LIN {X 0,Y 255.736,Z 943.824,A -85,B 0,C 180,E1 11654.094,E2 11654.094} C_VEL
LIN {X 0,Y 247.335,Z 955.504,A -85,B 0,C 180,E1 11649.69,E2 11649.69} C_VEL
LIN {X 0,Y 239.94,Z 965.687,A -85,B 0,C 180,E1 11644.807,E2 11644.807} C_VEL
LIN {X 0,Y 233.834,Z 974.598,A -85,B 0,C 180,E1 11639.45,E2 11639.45} C_VEL
LIN {X 0,Y 229.531,Z 981.362,A -85,B 0,C 180,E1 11634.168,E2 11634.168} C_VEL
LIN {X 0,Y 226.431,Z 987.137,A -85,B 0,C 180,E1 11628.268,E2 11628.268} C_VEL
LIN {X 0,Y 224.909,Z 990.729,A -85,B 0,C 180,E1 11623.102,E2 11623.102} C_VEL
LIN {X 0,Y 224.206,Z 993.296,A -85,B 0,C 180,E1 11617.687,E2 11617.687} C_VEL
LIN {X 0,Y 224.031,Z 994.4,A -85,B 0,C 180,E1 11612.557,E2 11612.557} C_VEL
LIN {X 0,Y 224.032,Z 994.473,A -85,B 0,C 180,E1 11608.209,E2 11608.209} C_VEL
LIN {X 0,Y 224.138,Z 993.662,A -85,B 0,C 180,E1 11603.597,E2 11603.597} C_VEL
LIN {X 0,Y 224.657,Z 991.562,A -85,B 0,C 180,E1 11598.187,E2 11598.187} C_VEL
LIN {X 0,Y 226.005,Z 988.015,A -85,B 0,C 180,E1 11592.759,E2 11592.759} C_VEL
LIN {X 0,Y 228.675,Z 982.95,A -85,B 0,C 180,E1 11587.101,E2 11587.101} C_VEL
LIN {X 0,Y 232.823,Z 976.112,A -85,B 0,C 180,E1 11581.533,E2 11581.533} C_VEL
LIN {X 0,Y 238.787,Z 967.412,A -85,B 0,C 180,E1 11576.004,E2 11576.004} C_VEL
LIN {X 0,Y 245.71,Z 957.743,A -85,B 0,C 180,E1 11571.2,E2 11571.2} C_VEL
LIN {X 0,Y 254.271,Z 945.935,A -85,B 0,C 180,E1 11566.522,E2 11566.522} C_VEL
LIN {X 0,Y 263.274,Z 933.388,A -85,B 0,C 180,E1 11562.533,E2 11562.533} C_VEL
LIN {X 0,Y 272.73,Z 919.575,A -85,B 0,C 180,E1 11559.001,E2 11559.001} C_VEL
LIN {X 0,Y 282.527,Z 904.622,A -85,B 0,C 180,E1 11555.871,E2 11555.871} C_VEL
LIN {X 0,Y 292.626,Z 887.873,A -85,B 0,C 180,E1 11553.047,E2 11553.047} C_VEL
LIN {X 0,Y 302.589,Z 870.047,A -85,B 0,C 180,E1 11550.589,E2 11550.589} C_VEL
LIN {X 0,Y 311.686,Z 851.804,A -85,B 0,C 180,E1 11548.554,E2 11548.554} C_VEL
LIN {X 0,Y 320.677,Z 831.7,A -85,B 0,C 180,E1 11546.722,E2 11546.722} C_VEL
LIN {X 0,Y 327.973,Z 812.96,A -85,B 0,C 180,E1 11545.336,E2 11545.336} C_VEL
LIN {X 0,Y 335.436,Z 790.655,A -85,B 0,C 180,E1 11544.005,E2 11544.005} C_VEL
LIN {X 0,Y 338.946,Z 778.487,A -85,B 0,C 180,E1 11543.397,E2 11543.397} C_VEL
LIN {X 0,Y 340.411,Z 771.364,A -85,B 0,C 180,E1 11542.929,E2 11542.929} C_VEL
LIN {X 0,Y 342.304,Z 753.795,A -85,B 0,C 180,E1 11541.314,E2 11541.314} C_VEL
LIN {X 0,Y 343.393,Z 746.488,A -85,B 0,C 180,E1 11540.937,E2 11540.937} C_VEL
LIN {X 0,Y 347.214,Z 723.354,A -85,B 0,C 180,E1 11540.335,E2 11540.335} C_VEL
LIN {X 0,Y 352.658,Z 665.576,A -85,B 0,C 180,E1 11539.208,E2 11539.208} C_VEL
LIN {X 0,Y 362.376,Z 558.402,A -85,B 0,C 180,E1 11537.172,E2 11537.172} C_VEL
LIN {X 0,Y 358.498,Z 551.455,A -85,B 0,C 180,E1 11534.455,E2 11534.455} C_VEL
LIN {X 0,Y 356.299,Z 547.697,A -85,B 0,C 180,E1 11532.644,E2 11532.644} C_VEL
LIN {X 0,Y 354.33,Z 544.268,A -85,B 0,C 180,E1 11530.734,E2 11530.734} C_VEL
LIN {X 0,Y 352.104,Z 540.388,A -85,B 0,C 180,E1 11527.999,E2 11527.999} C_VEL
LIN {X 0,Y 349.943,Z 536.182,A -85,B 0,C 180,E1 11523.44,E2 11523.44} C_VEL
LIN {X 0,Y 349.775,Z 535.565,A -85,B 0,C 180,E1 11522.622,E2 11522.622} C_VEL
LIN {X 0,Y 349.881,Z 535.803,A -85,B 0,C 180,E1 11517.38,E2 11517.38} C_VEL
LIN {X 0,Y 351.533,Z 539.751,A -85,B 0,C 180,E1 11513.304,E2 11513.304} C_VEL
LIN {X 0,Y 352.499,Z 541.08,A -85,B 0,C 180,E1 11511.929,E2 11511.929} C_VEL
LIN {X 0,Y 355.346,Z 546.022,A -85,B 0,C 180,E1 11508.723,E2 11508.723} C_VEL
LIN {X 0,Y 358.175,Z 550.942,A -85,B 0,C 180,E1 11506.274,E2 11506.274} C_VEL
LIN {X 0,Y 361.653,Z 557.016,A -85,B 0,C 180,E1 11503.786,E2 11503.786} C_VEL
LIN {X 0,Y 362.516,Z 559.023,A -85,B 0,C 180,E1 11503.197,E2 11503.197} C_VEL
LIN {X 0,Y 346.966,Z 729.479,A -85,B 0,C 180,E1 11499.934,E2 11499.934} C_VEL
LIN {X 0,Y 343.166,Z 753.522,A -85,B 0,C 180,E1 11499.355,E2 11499.355} C_VEL
LIN {X 0,Y 338.384,Z 775.393,A -85,B 0,C 180,E1 11498.689,E2 11498.689} C_VEL
LIN {X 0,Y 332.181,Z 797.399,A -85,B 0,C 180,E1 11497.784,E2 11497.784} C_VEL
LIN {X 0,Y 325.416,Z 817.772,A -85,B 0,C 180,E1 11496.722,E2 11496.722} C_VEL
LIN {X 0,Y 317.319,Z 838.274,A -85,B 0,C 180,E1 11495.361,E2 11495.361} C_VEL
LIN {X 0,Y 308.383,Z 858.36,A -85,B 0,C 180,E1 11493.712,E2 11493.712} C_VEL
LIN {X 0,Y 298.925,Z 877.022,A -85,B 0,C 180,E1 11491.796,E2 11491.796} C_VEL
LIN {X 0,Y 288.539,Z 895.73,A -85,B 0,C 180,E1 11489.432,E2 11489.432} C_VEL
LIN {X 0,Y 278.676,Z 911.928,A -85,B 0,C 180,E1 11486.896,E2 11486.896} C_VEL
LIN {X 0,Y 267.229,Z 929.456,A -85,B 0,C 180,E1 11483.494,E2 11483.494} C_VEL
LIN {X 0,Y 257.227,Z 944.006,A -85,B 0,C 180,E1 11479.967,E2 11479.967} C_VEL
LIN {X 0,Y 247.666,Z 957.322,A -85,B 0,C 180,E1 11475.934,E2 11475.934} C_VEL
LIN {X 0,Y 238.916,Z 969.495,A -85,B 0,C 180,E1 11471.388,E2 11471.388} C_VEL
LIN {X 0,Y 231.282,Z 980.172,A -85,B 0,C 180,E1 11466.314,E2 11466.314} C_VEL
LIN {X 0,Y 225.037,Z 989.575,A -85,B 0,C 180,E1 11460.724,E2 11460.724} C_VEL
LIN {X 0,Y 220.731,Z 996.778,A -85,B 0,C 180,E1 11455.199,E2 11455.199} C_VEL
LIN {X 0,Y 217.753,Z 1003.039,A -85,B 0,C 180,E1 11448.937,E2 11448.937} C_VEL
LIN {X 0,Y 216.47,Z 1006.872,A -85,B 0,C 180,E1 11443.624,E2 11443.624} C_VEL
LIN {X 0,Y 216.012,Z 1009.708,A -85,B 0,C 180,E1 11437.89,E2 11437.89} C_VEL
LIN {X 0,Y 216.005,Z 1010.89,A -85,B 0,C 180,E1 11432.654,E2 11432.654} C_VEL
LIN {X 0,Y 216.025,Z 1010.985,A -85,B 0,C 180,E1 11428.41,E2 11428.41} C_VEL
LIN {X 0,Y 216,Z 1010.188,A -85,B 0,C 180,E1 11423.89,E2 11423.89} C_VEL
LIN {X 0,Y 216.179,Z 1008.237,A -85,B 0,C 180,E1 11418.801,E2 11418.801} C_VEL
LIN {X 0,Y 217.196,Z 1004.462,A -85,B 0,C 180,E1 11412.868,E2 11412.868} C_VEL
LIN {X 0,Y 219.243,Z 999.668,A -85,B 0,C 180,E1 11407.479,E2 11407.479} C_VEL
LIN {X 0,Y 223.42,Z 992.094,A -85,B 0,C 180,E1 11401.102,E2 11401.102} C_VEL
LIN {X 0,Y 228.818,Z 983.779,A -85,B 0,C 180,E1 11395.675,E2 11395.675} C_VEL
LIN {X 0,Y 235.817,Z 973.673,A -85,B 0,C 180,E1 11390.504,E2 11390.504} C_VEL
LIN {X 0,Y 244.436,Z 961.795,A -85,B 0,C 180,E1 11385.623,E2 11385.623} C_VEL
LIN {X 0,Y 253.552,Z 949.029,A -85,B 0,C 180,E1 11381.483,E2 11381.483} C_VEL
LIN {X 0,Y 264.051,Z 934.069,A -85,B 0,C 180,E1 11377.563,E2 11377.563} C_VEL
LIN {X 0,Y 274.249,Z 918.722,A -85,B 0,C 180,E1 11374.344,E2 11374.344} C_VEL
LIN {X 0,Y 285.492,Z 900.645,A -85,B 0,C 180,E1 11371.303,E2 11371.303} C_VEL
LIN {X 0,Y 295.736,Z 882.842,A -85,B 0,C 180,E1 11368.89,E2 11368.89} C_VEL
LIN {X 0,Y 305.363,Z 864.194,A -85,B 0,C 180,E1 11366.862,E2 11366.862} C_VEL
LIN {X 0,Y 314.652,Z 844.373,A -85,B 0,C 180,E1 11365.106,E2 11365.106} C_VEL
LIN {X 0,Y 322.658,Z 824.612,A -85,B 0,C 180,E1 11363.711,E2 11363.711} C_VEL
LIN {X 0,Y 330.096,Z 803.74,A -85,B 0,C 180,E1 11362.523,E2 11362.523} C_VEL
LIN {X 0,Y 336.468,Z 781.982,A -85,B 0,C 180,E1 11361.564,E2 11361.564} C_VEL
LIN {X 0,Y 342.107,Z 758.231,A -85,B 0,C 180,E1 11360.78,E2 11360.78} C_VEL
LIN {X 0,Y 345.954,Z 736.026,A -85,B 0,C 180,E1 11360.221,E2 11360.221} C_VEL
LIN {X 0,Y 349.308,Z 704.022,A -85,B 0,C 180,E1 11359.57,E2 11359.57} C_VEL
LIN {X 0,Y 362.363,Z 558.559,A -85,B 0,C 180,E1 11356.783,E2 11356.783} C_VEL
LIN {X 0,Y 358.527,Z 551.667,A -85,B 0,C 180,E1 11354.123,E2 11354.123} C_VEL
LIN {X 0,Y 356.027,Z 547.407,A -85,B 0,C 180,E1 11352.076,E2 11352.076} C_VEL
LIN {X 0,Y 354.212,Z 544.29,A -85,B 0,C 180,E1 11350.325,E2 11350.325} C_VEL
LIN {X 0,Y 351.903,Z 540.251,A -85,B 0,C 180,E1 11347.51,E2 11347.51} C_VEL
LIN {X 0,Y 349.816,Z 536.268,A -85,B 0,C 180,E1 11343.277,E2 11343.277} C_VEL
LIN {X 0,Y 349.633,Z 535.518,A -85,B 0,C 180,E1 11342.458,E2 11342.458} C_VEL
LIN {X 0,Y 349.699,Z 535.594,A -85,B 0,C 180,E1 11336.721,E2 11336.721} C_VEL
LIN {X 0,Y 351.727,Z 540.075,A -85,B 0,C 180,E1 11332.157,E2 11332.157} C_VEL
LIN {X 0,Y 352.494,Z 541.282,A -85,B 0,C 180,E1 11331.107,E2 11331.107} C_VEL
LIN {X 0,Y 355.101,Z 545.709,A -85,B 0,C 180,E1 11328.221,E2 11328.221} C_VEL
LIN {X 0,Y 357.925,Z 550.622,A -85,B 0,C 180,E1 11325.769,E2 11325.769} C_VEL
LIN {X 0,Y 361.629,Z 557.156,A -85,B 0,C 180,E1 11323.123,E2 11323.123} C_VEL
LIN {X 0,Y 362.217,Z 558.605,A -85,B 0,C 180,E1 11322.717,E2 11322.717} C_VEL
LIN {X 0,Y 347.375,Z 720.612,A -85,B 0,C 180,E1 11319.623,E2 11319.623} C_VEL
LIN {X 0,Y 343.68,Z 744.239,A -85,B 0,C 180,E1 11319.029,E2 11319.029} C_VEL
LIN {X 0,Y 339.3,Z 764.96,A -85,B 0,C 180,E1 11318.331,E2 11318.331} C_VEL
LIN {X 0,Y 333.531,Z 786.231,A -85,B 0,C 180,E1 11317.399,E2 11317.399} C_VEL
LIN {X 0,Y 327.011,Z 806.35,A -85,B 0,C 180,E1 11316.295,E2 11316.295} C_VEL
LIN {X 0,Y 319.097,Z 826.901,A -85,B 0,C 180,E1 11314.883,E2 11314.883} C_VEL
LIN {X 0,Y 310.299,Z 846.954,A -85,B 0,C 180,E1 11313.183,E2 11313.183} C_VEL
LIN {X 0,Y 300.712,Z 865.928,A -85,B 0,C 180,E1 11311.176,E2 11311.176} C_VEL
LIN {X 0,Y 290.328,Z 884.559,A -85,B 0,C 180,E1 11308.752,E2 11308.752} C_VEL
LIN {X 0,Y 280.707,Z 900.187,A -85,B 0,C 180,E1 11306.243,E2 11306.243} C_VEL
LIN {X 0,Y 269.499,Z 917.069,A -85,B 0,C 180,E1 11302.898,E2 11302.898} C_VEL
LIN {X 0,Y 259.975,Z 930.527,A -85,B 0,C 180,E1 11299.588,E2 11299.588} C_VEL
LIN {X 0,Y 249.862,Z 944.136,A -85,B 0,C 180,E1 11295.414,E2 11295.414} C_VEL
LIN {X 0,Y 241.023,Z 955.816,A -85,B 0,C 180,E1 11290.947,E2 11290.947} C_VEL
LIN {X 0,Y 233.193,Z 965.999,A -85,B 0,C 180,E1 11285.968,E2 11285.968} C_VEL
LIN {X 0,Y 226.678,Z 974.909,A -85,B 0,C 180,E1 11280.476,E2 11280.476} C_VEL
LIN {X 0,Y 222.049,Z 981.671,A -85,B 0,C 180,E1 11275.037,E2 11275.037} C_VEL
LIN {X 0,Y 218.63,Z 987.551,A -85,B 0,C 180,E1 11268.795,E2 11268.795} C_VEL
LIN {X 0,Y 216.959,Z 991.187,A -85,B 0,C 180,E1 11263.32,E2 11263.32} C_VEL
LIN {X 0,Y 216.2,Z 993.743,A -85,B 0,C 180,E1 11257.439,E2 11257.439} C_VEL
LIN {X 0,Y 216.037,Z 994.721,A -85,B 0,C 180,E1 11252.386,E2 11252.386} C_VEL
LIN {X 0,Y 216.04,Z 994.751,A -85,B 0,C 180,E1 11247.878,E2 11247.878} C_VEL
LIN {X 0,Y 216.183,Z 993.835,A -85,B 0,C 180,E1 11242.826,E2 11242.826} C_VEL
LIN {X 0,Y 216.884,Z 991.406,A -85,B 0,C 180,E1 11236.945,E2 11236.945} C_VEL
LIN {X 0,Y 218.436,Z 987.924,A -85,B 0,C 180,E1 11231.59,E2 11231.59} C_VEL
LIN {X 0,Y 221.816,Z 982.087,A -85,B 0,C 180,E1 11225.218,E2 11225.218} C_VEL
LIN {X 0,Y 226.35,Z 975.393,A -85,B 0,C 180,E1 11219.766,E2 11219.766} C_VEL
LIN {X 0,Y 232.77,Z 966.624,A -85,B 0,C 180,E1 11214.258,E2 11214.258} C_VEL
LIN {X 0,Y 240.508,Z 956.545,A -85,B 0,C 180,E1 11209.26,E2 11209.26} C_VEL
LIN {X 0,Y 249.27,Z 944.999,A -85,B 0,C 180,E1 11204.773,E2 11204.773} C_VEL
LIN {X 0,Y 258.88,Z 932.201,A -85,B 0,C 180,E1 11200.748,E2 11200.748} C_VEL
LIN {X 0,Y 268.781,Z 918.217,A -85,B 0,C 180,E1 11197.251,E2 11197.251} C_VEL
LIN {X 0,Y 279.669,Z 902.002,A -85,B 0,C 180,E1 11193.968,E2 11193.968} C_VEL
LIN {X 0,Y 289.343,Z 886.364,A -85,B 0,C 180,E1 11191.411,E2 11191.411} C_VEL
LIN {X 0,Y 300.212,Z 867.107,A -85,B 0,C 180,E1 11188.856,E2 11188.856} C_VEL
LIN {X 0,Y 309.44,Z 848.964,A -85,B 0,C 180,E1 11186.911,E2 11186.911} C_VEL
LIN {X 0,Y 318.223,Z 829.319,A -85,B 0,C 180,E1 11185.203,E2 11185.203} C_VEL
LIN {X 0,Y 325.744,Z 810.262,A -85,B 0,C 180,E1 11183.851,E2 11183.851} C_VEL
LIN {X 0,Y 332.859,Z 788.912,A -85,B 0,C 180,E1 11182.635,E2 11182.635} C_VEL
LIN {X 0,Y 338.464,Z 768.92,A -85,B 0,C 180,E1 11181.725,E2 11181.725} C_VEL
LIN {X 0,Y 343.393,Z 746.488,A -85,B 0,C 180,E1 11180.937,E2 11180.937} C_VEL
LIN {X 0,Y 344.514,Z 739.093,A -85,B 0,C 180,E1 11180.585,E2 11180.585} C_VEL
LIN {X 0,Y 345.183,Z 720.8,A -85,B 0,C 180,E1 11179.191,E2 11179.191} C_VEL
LIN {X 0,Y 345.682,Z 713.298,A -85,B 0,C 180,E1 11178.876,E2 11178.876} C_VEL
LIN {X 0,Y 359.612,Z 563.719,A -85,B 0,C 180,E1 11176.046,E2 11176.046} C_VEL
LIN {X 0,Y 355.587,Z 556.366,A -85,B 0,C 180,E1 11172.918,E2 11172.918} C_VEL
LIN {X 0,Y 352.966,Z 551.864,A -85,B 0,C 180,E1 11170.363,E2 11170.363} C_VEL
LIN {X 0,Y 350.894,Z 548.153,A -85,B 0,C 180,E1 11167.697,E2 11167.697} C_VEL
LIN {X 0,Y 348.892,Z 543.886,A -85,B 0,C 180,E1 11163.122,E2 11163.122} C_VEL
LIN {X 0,Y 348.663,Z 543.461,A -85,B 0,C 180,E1 11161.972,E2 11161.972} C_VEL
LIN {X 0,Y 348.864,Z 543.694,A -85,B 0,C 180,E1 11157.536,E2 11157.536} C_VEL
LIN {X 0,Y 350.453,Z 547.629,A -85,B 0,C 180,E1 11153.447,E2 11153.447} C_VEL
LIN {X 0,Y 351.334,Z 548.905,A -85,B 0,C 180,E1 11152.149,E2 11152.149} C_VEL
LIN {X 0,Y 354.024,Z 553.722,A -85,B 0,C 180,E1 11149.01,E2 11149.01} C_VEL
LIN {X 0,Y 356.874,Z 558.835,A -85,B 0,C 180,E1 11146.471,E2 11146.471} C_VEL
LIN {X 0,Y 359.77,Z 564.022,A -85,B 0,C 180,E1 11144.326,E2 11144.326} C_VEL
LIN {X 0,Y 344.288,Z 729.198,A -85,B 0,C 180,E1 11141.191,E2 11141.191} C_VEL
LIN {X 0,Y 340.425,Z 753.168,A -85,B 0,C 180,E1 11140.625,E2 11140.625} C_VEL
LIN {X 0,Y 335.387,Z 775.727,A -85,B 0,C 180,E1 11139.951,E2 11139.951} C_VEL
LIN {X 0,Y 328.992,Z 797.784,A -85,B 0,C 180,E1 11139.057,E2 11139.057} C_VEL
LIN {X 0,Y 321.945,Z 818.389,A -85,B 0,C 180,E1 11137.995,E2 11137.995} C_VEL
LIN {X 0,Y 314.004,Z 837.972,A -85,B 0,C 180,E1 11136.715,E2 11136.715} C_VEL
LIN {X 0,Y 304.795,Z 858.143,A -85,B 0,C 180,E1 11135.086,E2 11135.086} C_VEL
LIN {X 0,Y 295.23,Z 876.513,A -85,B 0,C 180,E1 11133.229,E2 11133.229} C_VEL
LIN {X 0,Y 284.769,Z 894.861,A -85,B 0,C 180,E1 11130.948,E2 11130.948} C_VEL
LIN {X 0,Y 274.559,Z 911.107,A -85,B 0,C 180,E1 11128.437,E2 11128.437} C_VEL
LIN {X 0,Y 263.06,Z 928.159,A -85,B 0,C 180,E1 11125.175,E2 11125.175} C_VEL
LIN {X 0,Y 253.036,Z 942.127,A -85,B 0,C 180,E1 11121.837,E2 11121.837} C_VEL
LIN {X 0,Y 242.401,Z 956.361,A -85,B 0,C 180,E1 11117.584,E2 11117.584} C_VEL
LIN {X 0,Y 233.106,Z 968.597,A -85,B 0,C 180,E1 11112.995,E2 11112.995} C_VEL
LIN {X 0,Y 224.931,Z 979.388,A -85,B 0,C 180,E1 11107.834,E2 11107.834} C_VEL
LIN {X 0,Y 218.164,Z 988.898,A -85,B 0,C 180,E1 11102.113,E2 11102.113} C_VEL
LIN {X 0,Y 213.429,Z 996.154,A -85,B 0,C 180,E1 11096.424,E2 11096.424} C_VEL
LIN {X 0,Y 210.206,Z 1002.23,A -85,B 0,C 180,E1 11090.316,E2 11090.316} C_VEL
LIN {X 0,Y 208.596,Z 1006.399,A -85,B 0,C 180,E1 11084.432,E2 11084.432} C_VEL
LIN {X 0,Y 208.058,Z 1009.14,A -85,B 0,C 180,E1 11078.846,E2 11078.846} C_VEL
LIN {X 0,Y 208,Z 1010.54,A -85,B 0,C 180,E1 11073.307,E2 11073.307} C_VEL
LIN {X 0,Y 208.03,Z 1010.706,A -85,B 0,C 180,E1 11068.593,E2 11068.593} C_VEL
LIN {X 0,Y 208.003,Z 1009.958,A -85,B 0,C 180,E1 11063.931,E2 11063.931} C_VEL
LIN {X 0,Y 208.143,Z 1008.293,A -85,B 0,C 180,E1 11059.204,E2 11059.204} C_VEL
LIN {X 0,Y 209.127,Z 1004.799,A -85,B 0,C 180,E1 11053.046,E2 11053.046} C_VEL
LIN {X 0,Y 211.328,Z 999.885,A -85,B 0,C 180,E1 11047.175,E2 11047.175} C_VEL
LIN {X 0,Y 215.468,Z 992.874,A -85,B 0,C 180,E1 11040.845,E2 11040.845} C_VEL
LIN {X 0,Y 220.996,Z 984.741,A -85,B 0,C 180,E1 11035.251,E2 11035.251} C_VEL
LIN {X 0,Y 228.997,Z 973.899,A -85,B 0,C 180,E1 11029.422,E2 11029.422} C_VEL
LIN {X 0,Y 237.623,Z 962.61,A -85,B 0,C 180,E1 11024.643,E2 11024.643} C_VEL
LIN {X 0,Y 247.548,Z 949.427,A -85,B 0,C 180,E1 11020.246,E2 11020.246} C_VEL
LIN {X 0,Y 258.234,Z 934.926,A -85,B 0,C 180,E1 11016.365,E2 11016.365} C_VEL
LIN {X 0,Y 268.996,Z 919.346,A -85,B 0,C 180,E1 11013.063,E2 11013.063} C_VEL
LIN {X 0,Y 280.592,Z 901.455,A -85,B 0,C 180,E1 11010.027,E2 11010.027} C_VEL
LIN {X 0,Y 290.757,Z 884.374,A -85,B 0,C 180,E1 11007.701,E2 11007.701} C_VEL
LIN {X 0,Y 301.381,Z 864.601,A -85,B 0,C 180,E1 11005.542,E2 11005.542} C_VEL
LIN {X 0,Y 310.762,Z 845.178,A -85,B 0,C 180,E1 11003.832,E2 11003.832} C_VEL
LIN {X 0,Y 319.352,Z 824.613,A -85,B 0,C 180,E1 11002.395,E2 11002.395} C_VEL
LIN {X 0,Y 327.079,Z 803.428,A -85,B 0,C 180,E1 11001.212,E2 11001.212} C_VEL
LIN {X 0,Y 333.585,Z 781.67,A -85,B 0,C 180,E1 11000.275,E2 11000.275} C_VEL
LIN {X 0,Y 339.361,Z 757.786,A -85,B 0,C 180,E1 10999.506,E2 10999.506} C_VEL
LIN {X 0,Y 343.28,Z 735.546,A -85,B 0,C 180,E1 10998.956,E2 10998.956} C_VEL
LIN {X 0,Y 346.729,Z 703.302,A -85,B 0,C 180,E1 10998.308,E2 10998.308} C_VEL
LIN {X 0,Y 359.572,Z 563.811,A -85,B 0,C 180,E1 10995.648,E2 10995.648} C_VEL
LIN {X 0,Y 355.496,Z 556.371,A -85,B 0,C 180,E1 10992.507,E2 10992.507} C_VEL
LIN {X 0,Y 352.919,Z 551.985,A -85,B 0,C 180,E1 10990.034,E2 10990.034} C_VEL
LIN {X 0,Y 350.809,Z 548.129,A -85,B 0,C 180,E1 10987.368,E2 10987.368} C_VEL
LIN {X 0,Y 348.787,Z 544.163,A -85,B 0,C 180,E1 10983.122,E2 10983.122} C_VEL
LIN {X 0,Y 348.614,Z 543.445,A -85,B 0,C 180,E1 10982.301,E2 10982.301} C_VEL
LIN {X 0,Y 348.68,Z 543.493,A -85,B 0,C 180,E1 10976.876,E2 10976.876} C_VEL
LIN {X 0,Y 350.754,Z 548.075,A -85,B 0,C 180,E1 10972.135,E2 10972.135} C_VEL
LIN {X 0,Y 353.703,Z 553.253,A -85,B 0,C 180,E1 10968.587,E2 10968.587} C_VEL
LIN {X 0,Y 356.528,Z 558.35,A -85,B 0,C 180,E1 10966.043,E2 10966.043} C_VEL
LIN {X 0,Y 359.461,Z 563.796,A -85,B 0,C 180,E1 10963.843,E2 10963.843} C_VEL
LIN {X 0,Y 344.671,Z 720.935,A -85,B 0,C 180,E1 10960.869,E2 10960.869} C_VEL
LIN {X 0,Y 340.897,Z 744.553,A -85,B 0,C 180,E1 10960.285,E2 10960.285} C_VEL
LIN {X 0,Y 336.421,Z 765.272,A -85,B 0,C 180,E1 10959.601,E2 10959.601} C_VEL
LIN {X 0,Y 330.525,Z 786.54,A -85,B 0,C 180,E1 10958.686,E2 10958.686} C_VEL
LIN {X 0,Y 323.854,Z 806.66,A -85,B 0,C 180,E1 10957.601,E2 10957.601} C_VEL
LIN {X 0,Y 315.75,Z 827.211,A -85,B 0,C 180,E1 10956.211,E2 10956.211} C_VEL
LIN {X 0,Y 306.724,Z 847.263,A -85,B 0,C 180,E1 10954.535,E2 10954.535} C_VEL
LIN {X 0,Y 296.818,Z 866.336,A -85,B 0,C 180,E1 10952.541,E2 10952.541} C_VEL
LIN {X 0,Y 286.325,Z 884.625,A -85,B 0,C 180,E1 10950.188,E2 10950.188} C_VEL
LIN {X 0,Y 276.269,Z 900.441,A -85,B 0,C 180,E1 10947.668,E2 10947.668} C_VEL
LIN {X 0,Y 264.62,Z 917.38,A -85,B 0,C 180,E1 10944.318,E2 10944.318} C_VEL
LIN {X 0,Y 254.707,Z 930.839,A -85,B 0,C 180,E1 10941.001,E2 10941.001} C_VEL
LIN {X 0,Y 244.125,Z 944.448,A -85,B 0,C 180,E1 10936.797,E2 10936.797} C_VEL
LIN {X 0,Y 234.565,Z 956.47,A -85,B 0,C 180,E1 10932.124,E2 10932.124} C_VEL
LIN {X 0,Y 226.193,Z 966.758,A -85,B 0,C 180,E1 10926.948,E2 10926.948} C_VEL
LIN {X 0,Y 219.053,Z 975.904,A -85,B 0,C 180,E1 10921.045,E2 10921.045} C_VEL
LIN {X 0,Y 214.235,Z 982.567,A -85,B 0,C 180,E1 10915.424,E2 10915.424} C_VEL
LIN {X 0,Y 210.737,Z 988.147,A -85,B 0,C 180,E1 10909.107,E2 10909.107} C_VEL
LIN {X 0,Y 209.013,Z 991.644,A -85,B 0,C 180,E1 10903.554,E2 10903.554} C_VEL
LIN {X 0,Y 208.208,Z 994.109,A -85,B 0,C 180,E1 10897.448,E2 10897.448} C_VEL
LIN {X 0,Y 208.043,Z 995.021,A -85,B 0,C 180,E1 10892.478,E2 10892.478} C_VEL
LIN {X 0,Y 208.044,Z 995.051,A -85,B 0,C 180,E1 10887.796,E2 10887.796} C_VEL
LIN {X 0,Y 208.191,Z 994.2,A -85,B 0,C 180,E1 10882.827,E2 10882.827} C_VEL
LIN {X 0,Y 208.88,Z 992.015,A -85,B 0,C 180,E1 10876.999,E2 10876.999} C_VEL
LIN {X 0,Y 210.587,Z 988.428,A -85,B 0,C 180,E1 10871.165,E2 10871.165} C_VEL
LIN {X 0,Y 213.994,Z 982.98,A -85,B 0,C 180,E1 10864.84,E2 10864.84} C_VEL
LIN {X 0,Y 218.716,Z 976.386,A -85,B 0,C 180,E1 10859.205,E2 10859.205} C_VEL
LIN {X 0,Y 225.753,Z 967.38,A -85,B 0,C 180,E1 10853.283,E2 10853.283} C_VEL
LIN {X 0,Y 233.443,Z 957.859,A -85,B 0,C 180,E1 10848.409,E2 10848.409} C_VEL
LIN {X 0,Y 243.022,Z 945.929,A -85,B 0,C 180,E1 10843.611,E2 10843.611} C_VEL
LIN {X 0,Y 253.164,Z 933.047,A -85,B 0,C 180,E1 10839.484,E2 10839.484} C_VEL
LIN {X 0,Y 263.881,Z 918.523,A -85,B 0,C 180,E1 10835.829,E2 10835.829} C_VEL
LIN {X 0,Y 275.167,Z 902.307,A -85,B 0,C 180,E1 10832.551,E2 10832.551} C_VEL
LIN {X 0,Y 285.165,Z 886.667,A -85,B 0,C 180,E1 10830.009,E2 10830.009} C_VEL
LIN {X 0,Y 296.364,Z 867.408,A -85,B 0,C 180,E1 10827.476,E2 10827.476} C_VEL
LIN {X 0,Y 305.849,Z 849.264,A -85,B 0,C 180,E1 10825.554,E2 10825.554} C_VEL
LIN {X 0,Y 314.861,Z 829.617,A -85,B 0,C 180,E1 10823.87,E2 10823.87} C_VEL
LIN {X 0,Y 322.956,Z 809.561,A -85,B 0,C 180,E1 10822.475,E2 10822.475} C_VEL
LIN {X 0,Y 330.197,Z 788.07,A -85,B 0,C 180,E1 10821.289,E2 10821.289} C_VEL
LIN {X 0,Y 336.266,Z 766.6,A -85,B 0,C 180,E1 10820.349,E2 10820.349} C_VEL
LIN {X 0,Y 340.928,Z 745.163,A -85,B 0,C 180,E1 10819.633,E2 10819.633} C_VEL
LIN {X 0,Y 344.72,Z 721.844,A -85,B 0,C 180,E1 10819.05,E2 10819.05} C_VEL
LIN {X 0,Y 345.682,Z 713.298,A -85,B 0,C 180,E1 10818.876,E2 10818.876} C_VEL
LIN {X 0,Y 346.177,Z 705.769,A -85,B 0,C 180,E1 10818.575,E2 10818.575} C_VEL
LIN {X 0,Y 346.074,Z 686.167,A -85,B 0,C 180,E1 10817.216,E2 10817.216} C_VEL
LIN {X 0,Y 346.442,Z 679.68,A -85,B 0,C 180,E1 10816.971,E2 10816.971} C_VEL
LIN {X 0,Y 356.948,Z 569.278,A -85,B 0,C 180,E1 10814.897,E2 10814.897} C_VEL
LIN {X 0,Y 353.7,Z 563.225,A -85,B 0,C 180,E1 10812.158,E2 10812.158} C_VEL
LIN {X 0,Y 351.689,Z 559.561,A -85,B 0,C 180,E1 10810.07,E2 10810.07} C_VEL
LIN {X 0,Y 349.807,Z 556.031,A -85,B 0,C 180,E1 10807.556,E2 10807.556} C_VEL
LIN {X 0,Y 347.853,Z 551.589,A -85,B 0,C 180,E1 10802.801,E2 10802.801} C_VEL
LIN {X 0,Y 347.825,Z 551.442,A -85,B 0,C 180,E1 10797.859,E2 10797.859} C_VEL
LIN {X 0,Y 349.477,Z 555.634,A -85,B 0,C 180,E1 10793.429,E2 10793.429} C_VEL
LIN {X 0,Y 350.226,Z 556.864,A -85,B 0,C 180,E1 10792.289,E2 10792.289} C_VEL
LIN {X 0,Y 352.787,Z 561.578,A -85,B 0,C 180,E1 10789.219,E2 10789.219} C_VEL
LIN {X 0,Y 355.481,Z 566.551,A -85,B 0,C 180,E1 10786.748,E2 10786.748} C_VEL
LIN {X 0,Y 357.095,Z 569.815,A -85,B 0,C 180,E1 10785.455,E2 10785.455} C_VEL
LIN {X 0,Y 341.771,Z 728.983,A -85,B 0,C 180,E1 10782.467,E2 10782.467} C_VEL
LIN {X 0,Y 337.815,Z 753.006,A -85,B 0,C 180,E1 10781.909,E2 10781.909} C_VEL
LIN {X 0,Y 332.803,Z 775.066,A -85,B 0,C 180,E1 10781.266,E2 10781.266} C_VEL
LIN {X 0,Y 326.74,Z 795.771,A -85,B 0,C 180,E1 10780.461,E2 10780.461} C_VEL
LIN {X 0,Y 319.343,Z 817.176,A -85,B 0,C 180,E1 10779.401,E2 10779.401} C_VEL
LIN {X 0,Y 310.829,Z 837.76,A -85,B 0,C 180,E1 10778.091,E2 10778.091} C_VEL
LIN {X 0,Y 301.432,Z 857.84,A -85,B 0,C 180,E1 10776.5,E2 10776.5} C_VEL
LIN {X 0,Y 291.5,Z 876.412,A -85,B 0,C 180,E1 10774.652,E2 10774.652} C_VEL
LIN {X 0,Y 280.482,Z 895.116,A -85,B 0,C 180,E1 10772.345,E2 10772.345} C_VEL
LIN {X 0,Y 269.962,Z 911.312,A -85,B 0,C 180,E1 10769.851,E2 10769.851} C_VEL
LIN {X 0,Y 257.752,Z 928.707,A -85,B 0,C 180,E1 10766.505,E2 10766.505} C_VEL
LIN {X 0,Y 247.369,Z 942.599,A -85,B 0,C 180,E1 10763.152,E2 10763.152} C_VEL
LIN {X 0,Y 236.3,Z 956.696,A -85,B 0,C 180,E1 10758.859,E2 10758.859} C_VEL
LIN {X 0,Y 226.59,Z 968.869,A -85,B 0,C 180,E1 10754.197,E2 10754.197} C_VEL
LIN {X 0,Y 217.993,Z 979.546,A -85,B 0,C 180,E1 10748.926,E2 10748.926} C_VEL
LIN {X 0,Y 210.839,Z 988.95,A -85,B 0,C 180,E1 10743.046,E2 10743.046} C_VEL
LIN {X 0,Y 205.812,Z 996.157,A -85,B 0,C 180,E1 10737.169,E2 10737.169} C_VEL
LIN {X 0,Y 202.14,Z 1002.569,A -85,B 0,C 180,E1 10730.256,E2 10730.256} C_VEL
LIN {X 0,Y 200.587,Z 1006.428,A -85,B 0,C 180,E1 10724.431,E2 10724.431} C_VEL
LIN {X 0,Y 200.038,Z 1009.176,A -85,B 0,C 180,E1 10718.248,E2 10718.248} C_VEL
LIN {X 0,Y 200.01,Z 1010.289,A -85,B 0,C 180,E1 10712.866,E2 10712.866} C_VEL
LIN {X 0,Y 200.034,Z 1010.385,A -85,B 0,C 180,E1 10708.282,E2 10708.282} C_VEL
LIN {X 0,Y 200.009,Z 1009.656,A -85,B 0,C 180,E1 10703.687,E2 10703.687} C_VEL
LIN {X 0,Y 200.179,Z 1007.988,A -85,B 0,C 180,E1 10698.769,E2 10698.769} C_VEL
LIN {X 0,Y 201.292,Z 1004.491,A -85,B 0,C 180,E1 10692.365,E2 10692.365} C_VEL
LIN {X 0,Y 203.715,Z 999.573,A -85,B 0,C 180,E1 10686.271,E2 10686.271} C_VEL
LIN {X 0,Y 208.214,Z 992.56,A -85,B 0,C 180,E1 10679.725,E2 10679.725} C_VEL
LIN {X 0,Y 214.16,Z 984.425,A -85,B 0,C 180,E1 10673.972,E2 10673.972} C_VEL
LIN {X 0,Y 222.69,Z 973.583,A -85,B 0,C 180,E1 10668.017,E2 10668.017} C_VEL
LIN {X 0,Y 231.743,Z 962.362,A -85,B 0,C 180,E1 10663.193,E2 10663.193} C_VEL
LIN {X 0,Y 242.22,Z 949.111,A -85,B 0,C 180,E1 10658.733,E2 10658.733} C_VEL
LIN {X 0,Y 253.365,Z 934.609,A -85,B 0,C 180,E1 10654.842,E2 10654.842} C_VEL
LIN {X 0,Y 264.559,Z 919.013,A -85,B 0,C 180,E1 10651.548,E2 10651.548} C_VEL
LIN {X 0,Y 276.843,Z 900.663,A -85,B 0,C 180,E1 10648.472,E2 10648.472} C_VEL
LIN {X 0,Y 287.389,Z 883.446,A -85,B 0,C 180,E1 10646.169,E2 10646.169} C_VEL
LIN {X 0,Y 297.936,Z 864.289,A -85,B 0,C 180,E1 10644.118,E2 10644.118} C_VEL
LIN {X 0,Y 307.681,Z 844.605,A -85,B 0,C 180,E1 10642.42,E2 10642.42} C_VEL
LIN {X 0,Y 316.312,Z 824.382,A -85,B 0,C 180,E1 10641.038,E2 10641.038} C_VEL
LIN {X 0,Y 324.237,Z 803.117,A -85,B 0,C 180,E1 10639.878,E2 10639.878} C_VEL
LIN {X 0,Y 330.874,Z 781.358,A -85,B 0,C 180,E1 10638.963,E2 10638.963} C_VEL
LIN {X 0,Y 336.759,Z 757.472,A -85,B 0,C 180,E1 10638.215,E2 10638.215} C_VEL
LIN {X 0,Y 340.751,Z 735.228,A -85,B 0,C 180,E1 10637.676,E2 10637.676} C_VEL
LIN {X 0,Y 344.293,Z 702.888,A -85,B 0,C 180,E1 10637.034,E2 10637.034} C_VEL
LIN {X 0,Y 356.921,Z 569.404,A -85,B 0,C 180,E1 10634.52,E2 10634.52} C_VEL
LIN {X 0,Y 353.512,Z 563.08,A -85,B 0,C 180,E1 10631.667,E2 10631.667} C_VEL
LIN {X 0,Y 351.635,Z 559.68,A -85,B 0,C 180,E1 10629.74,E2 10629.74} C_VEL
LIN {X 0,Y 349.604,Z 555.883,A -85,B 0,C 180,E1 10627.064,E2 10627.064} C_VEL
LIN {X 0,Y 347.729,Z 551.865,A -85,B 0,C 180,E1 10622.801,E2 10622.801} C_VEL
LIN {X 0,Y 347.558,Z 551.359,A -85,B 0,C 180,E1 10621.978,E2 10621.978} C_VEL
LIN {X 0,Y 347.688,Z 551.588,A -85,B 0,C 180,E1 10616.867,E2 10616.867} C_VEL
LIN {X 0,Y 350.049,Z 556.661,A -85,B 0,C 180,E1 10611.706,E2 10611.706} C_VEL
LIN {X 0,Y 352.469,Z 561.116,A -85,B 0,C 180,E1 10608.795,E2 10608.795} C_VEL
LIN {X 0,Y 355.045,Z 565.897,A -85,B 0,C 180,E1 10606.399,E2 10606.399} C_VEL
LIN {X 0,Y 356.813,Z 569.323,A -85,B 0,C 180,E1 10604.98,E2 10604.98} C_VEL
LIN {X 0,Y 342.132,Z 721.258,A -85,B 0,C 180,E1 10602.135,E2 10602.135} C_VEL
LIN {X 0,Y 338.28,Z 744.866,A -85,B 0,C 180,E1 10601.562,E2 10601.562} C_VEL
LIN {X 0,Y 333.71,Z 765.584,A -85,B 0,C 180,E1 10600.892,E2 10600.892} C_VEL
LIN {X 0,Y 327.688,Z 786.85,A -85,B 0,C 180,E1 10599.996,E2 10599.996} C_VEL
LIN {X 0,Y 320.869,Z 806.969,A -85,B 0,C 180,E1 10598.932,E2 10598.932} C_VEL
LIN {X 0,Y 312.577,Z 827.52,A -85,B 0,C 180,E1 10597.567,E2 10597.567} C_VEL
LIN {X 0,Y 303.326,Z 847.572,A -85,B 0,C 180,E1 10595.918,E2 10595.918} C_VEL
LIN {X 0,Y 293.346,Z 866.299,A -85,B 0,C 180,E1 10593.993,E2 10593.993} C_VEL
LIN {X 0,Y 282.705,Z 884.387,A -85,B 0,C 180,E1 10591.708,E2 10591.708} C_VEL
LIN {X 0,Y 271.959,Z 900.769,A -85,B 0,C 180,E1 10589.125,E2 10589.125} C_VEL
LIN {X 0,Y 259.908,Z 917.692,A -85,B 0,C 180,E1 10585.791,E2 10585.791} C_VEL
LIN {X 0,Y 249.599,Z 931.15,A -85,B 0,C 180,E1 10582.472,E2 10582.472} C_VEL
LIN {X 0,Y 238.54,Z 944.761,A -85,B 0,C 180,E1 10578.245,E2 10578.245} C_VEL
LIN {X 0,Y 228.78,Z 956.441,A -85,B 0,C 180,E1 10573.664,E2 10573.664} C_VEL
LIN {X 0,Y 220.012,Z 966.623,A -85,B 0,C 180,E1 10568.5,E2 10568.5} C_VEL
LIN {X 0,Y 212.601,Z 975.531,A -85,B 0,C 180,E1 10562.736,E2 10562.736} C_VEL
LIN {X 0,Y 207.245,Z 982.291,A -85,B 0,C 180,E1 10556.965,E2 10556.965} C_VEL
LIN {X 0,Y 203.289,Z 988.059,A -85,B 0,C 180,E1 10550.436,E2 10550.436} C_VEL
LIN {X 0,Y 201.201,Z 991.796,A -85,B 0,C 180,E1 10544.385,E2 10544.385} C_VEL
LIN {X 0,Y 200.252,Z 994.347,A -85,B 0,C 180,E1 10538.035,E2 10538.035} C_VEL
LIN {X 0,Y 200.048,Z 995.321,A -85,B 0,C 180,E1 10532.577,E2 10532.577} C_VEL
LIN {X 0,Y 200.05,Z 995.372,A -85,B 0,C 180,E1 10527.994,E2 10527.994} C_VEL
LIN {X 0,Y 200.199,Z 994.565,A -85,B 0,C 180,E1 10522.827,E2 10522.827} C_VEL
LIN {X 0,Y 200.929,Z 992.472,A -85,B 0,C 180,E1 10516.768,E2 10516.768} C_VEL
LIN {X 0,Y 202.749,Z 988.931,A -85,B 0,C 180,E1 10510.708,E2 10510.708} C_VEL
LIN {X 0,Y 206.197,Z 983.851,A -85,B 0,C 180,E1 10504.413,E2 10504.413} C_VEL
LIN {X 0,Y 211.381,Z 977.037,A -85,B 0,C 180,E1 10498.332,E2 10498.332} C_VEL
LIN {X 0,Y 218.444,Z 968.583,A -85,B 0,C 180,E1 10492.504,E2 10492.504} C_VEL
LIN {X 0,Y 226.873,Z 958.67,A -85,B 0,C 180,E1 10487.263,E2 10487.263} C_VEL
LIN {X 0,Y 236.878,Z 946.859,A -85,B 0,C 180,E1 10482.388,E2 10482.388} C_VEL
LIN {X 0,Y 247.168,Z 934.346,A -85,B 0,C 180,E1 10478.307,E2 10478.307} C_VEL
LIN {X 0,Y 257.901,Z 920.493,A -85,B 0,C 180,E1 10474.732,E2 10474.732} C_VEL
LIN {X 0,Y 268.845,Z 905.535,A -85,B 0,C 180,E1 10471.616,E2 10471.616} C_VEL
LIN {X 0,Y 279.761,Z 889.163,A -85,B 0,C 180,E1 10468.892,E2 10468.892} C_VEL
LIN {X 0,Y 290.51,Z 871.669,A -85,B 0,C 180,E1 10466.523,E2 10466.523} C_VEL
LIN {X 0,Y 300.694,Z 852.906,A -85,B 0,C 180,E1 10464.493,E2 10464.493} C_VEL
LIN {X 0,Y 310.368,Z 832.936,A -85,B 0,C 180,E1 10462.742,E2 10462.742} C_VEL
LIN {X 0,Y 318.37,Z 813.847,A -85,B 0,C 180,E1 10461.397,E2 10461.397} C_VEL
LIN {X 0,Y 326.365,Z 791.535,A -85,B 0,C 180,E1 10460.132,E2 10460.132} C_VEL
LIN {X 0,Y 332.035,Z 772.449,A -85,B 0,C 180,E1 10459.275,E2 10459.275} C_VEL
LIN {X 0,Y 337.676,Z 748.701,A -85,B 0,C 180,E1 10458.447,E2 10458.447} C_VEL
LIN {X 0,Y 341.545,Z 726.722,A -85,B 0,C 180,E1 10457.883,E2 10457.883} C_VEL
LIN {X 0,Y 345.154,Z 693.391,A -85,B 0,C 180,E1 10457.228,E2 10457.228} C_VEL
LIN {X 0,Y 346.442,Z 679.68,A -85,B 0,C 180,E1 10456.971,E2 10456.971} C_VEL
LIN {X 0,Y 346.863,Z 672.143,A -85,B 0,C 180,E1 10456.668,E2 10456.668} C_VEL
LIN {X 0,Y 347.046,Z 652.551,A -85,B 0,C 180,E1 10455.312,E2 10455.312} C_VEL
LIN {X 0,Y 347.482,Z 646.068,A -85,B 0,C 180,E1 10455.072,E2 10455.072} C_VEL
LIN {X 0,Y 354.468,Z 574.884,A -85,B 0,C 180,E1 10453.76,E2 10453.76} C_VEL
LIN {X 0,Y 351.88,Z 570.048,A -85,B 0,C 180,E1 10451.39,E2 10451.39} C_VEL
LIN {X 0,Y 350.352,Z 567.151,A -85,B 0,C 180,E1 10449.694,E2 10449.694} C_VEL
LIN {X 0,Y 348.613,Z 563.792,A -85,B 0,C 180,E1 10447.25,E2 10447.25} C_VEL
LIN {X 0,Y 346.778,Z 559.365,A -85,B 0,C 180,E1 10442.314,E2 10442.314} C_VEL
LIN {X 0,Y 346.839,Z 559.477,A -85,B 0,C 180,E1 10437.853,E2 10437.853} C_VEL
LIN {X 0,Y 348.398,Z 563.511,A -85,B 0,C 180,E1 10433.574,E2 10433.574} C_VEL
LIN {X 0,Y 349.121,Z 564.816,A -85,B 0,C 180,E1 10432.43,E2 10432.43} C_VEL
LIN {X 0,Y 351.481,Z 569.275,A -85,B 0,C 180,E1 10429.511,E2 10429.511} C_VEL
LIN {X 0,Y 354.286,Z 574.603,A -85,B 0,C 180,E1 10426.869,E2 10426.869} C_VEL
LIN {X 0,Y 354.58,Z 575.378,A -85,B 0,C 180,E1 10426.605,E2 10426.605} C_VEL
LIN {X 0,Y 339.438,Z 728.661,A -85,B 0,C 180,E1 10423.763,E2 10423.763} C_VEL
LIN {X 0,Y 335.409,Z 752.687,A -85,B 0,C 180,E1 10423.217,E2 10423.217} C_VEL
LIN {X 0,Y 330.303,Z 774.774,A -85,B 0,C 180,E1 10422.59,E2 10422.59} C_VEL
LIN {X 0,Y 324.123,Z 795.475,A -85,B 0,C 180,E1 10421.809,E2 10421.809} C_VEL
LIN {X 0,Y 316.576,Z 816.878,A -85,B 0,C 180,E1 10420.777,E2 10420.777} C_VEL
LIN {X 0,Y 307.916,Z 837.372,A -85,B 0,C 180,E1 10419.506,E2 10419.506} C_VEL
LIN {X 0,Y 298.299,Z 857.462,A -85,B 0,C 180,E1 10417.951,E2 10417.951} C_VEL
LIN {X 0,Y 288.169,Z 875.934,A -85,B 0,C 180,E1 10416.151,E2 10416.151} C_VEL
LIN {X 0,Y 276.597,Z 895.024,A -85,B 0,C 180,E1 10413.832,E2 10413.832} C_VEL
LIN {X 0,Y 265.534,Z 911.517,A -85,B 0,C 180,E1 10411.314,E2 10411.314} C_VEL
LIN {X 0,Y 253.124,Z 928.559,A -85,B 0,C 180,E1 10408.042,E2 10408.042} C_VEL
LIN {X 0,Y 241.839,Z 943.072,A -85,B 0,C 180,E1 10404.527,E2 10404.527} C_VEL
LIN {X 0,Y 230.865,Z 956.383,A -85,B 0,C 180,E1 10400.428,E2 10400.428} C_VEL
LIN {X 0,Y 220.654,Z 968.556,A -85,B 0,C 180,E1 10395.715,E2 10395.715} C_VEL
LIN {X 0,Y 211.529,Z 979.232,A -85,B 0,C 180,E1 10390.354,E2 10390.354} C_VEL
LIN {X 0,Y 203.872,Z 988.637,A -85,B 0,C 180,E1 10384.329,E2 10384.329} C_VEL
LIN {X 0,Y 198.437,Z 995.845,A -85,B 0,C 180,E1 10378.268,E2 10378.268} C_VEL
LIN {X 0,Y 194.416,Z 1002.26,A -85,B 0,C 180,E1 10371.099,E2 10371.099} C_VEL
LIN {X 0,Y 192.711,Z 1006.033,A -85,B 0,C 180,E1 10365.199,E2 10365.199} C_VEL
LIN {X 0,Y 192.056,Z 1008.851,A -85,B 0,C 180,E1 10358.683,E2 10358.683} C_VEL
LIN {X 0,Y 192.013,Z 1009.989,A -85,B 0,C 180,E1 10352.985,E2 10352.985} C_VEL
LIN {X 0,Y 192.038,Z 1010.085,A -85,B 0,C 180,E1 10348.211,E2 10348.211} C_VEL
LIN {X 0,Y 192.009,Z 1009.354,A -85,B 0,C 180,E1 10343.423,E2 10343.423} C_VEL
LIN {X 0,Y 192.219,Z 1007.683,A -85,B 0,C 180,E1 10338.298,E2 10338.298} C_VEL
LIN {X 0,Y 193.481,Z 1004.182,A -85,B 0,C 180,E1 10331.628,E2 10331.628} C_VEL
LIN {X 0,Y 196.147,Z 999.262,A -85,B 0,C 180,E1 10325.296,E2 10325.296} C_VEL
LIN {X 0,Y 200.785,Z 992.61,A -85,B 0,C 180,E1 10318.814,E2 10318.814} C_VEL
LIN {X 0,Y 207.267,Z 984.315,A -85,B 0,C 180,E1 10312.745,E2 10312.745} C_VEL
LIN {X 0,Y 216.084,Z 973.794,A -85,B 0,C 180,E1 10306.786,E2 10306.786} C_VEL
LIN {X 0,Y 225.567,Z 962.632,A -85,B 0,C 180,E1 10301.876,E2 10301.876} C_VEL
LIN {X 0,Y 236.488,Z 949.508,A -85,B 0,C 180,E1 10297.368,E2 10297.368} C_VEL
LIN {X 0,Y 248.049,Z 935.132,A -85,B 0,C 180,E1 10293.458,E2 10293.458} C_VEL
LIN {X 0,Y 259.946,Z 919.186,A -85,B 0,C 180,E1 10290.08,E2 10290.08} C_VEL
LIN {X 0,Y 271.958,Z 901.951,A -85,B 0,C 180,E1 10287.176,E2 10287.176} C_VEL
LIN {X 0,Y 282.329,Z 885.593,A -85,B 0,C 180,E1 10284.974,E2 10284.974} C_VEL
LIN {X 0,Y 293.893,Z 865.46,A -85,B 0,C 180,E1 10282.801,E2 10282.801} C_VEL
LIN {X 0,Y 303.036,Z 847.564,A -85,B 0,C 180,E1 10281.254,E2 10281.254} C_VEL
LIN {X 0,Y 312.819,Z 825.701,A -85,B 0,C 180,E1 10279.748,E2 10279.748} C_VEL
LIN {X 0,Y 320.728,Z 805.157,A -85,B 0,C 180,E1 10278.632,E2 10278.632} C_VEL
LIN {X 0,Y 327.794,Z 782.944,A -85,B 0,C 180,E1 10277.699,E2 10277.699} C_VEL
LIN {X 0,Y 333.714,Z 760.164,A -85,B 0,C 180,E1 10276.981,E2 10276.981} C_VEL
LIN {X 0,Y 338.052,Z 737.028,A -85,B 0,C 180,E1 10276.424,E2 10276.424} C_VEL
LIN {X 0,Y 341.67,Z 706.223,A -85,B 0,C 180,E1 10275.813,E2 10275.813} C_VEL
LIN {X 0,Y 354.415,Z 574.964,A -85,B 0,C 180,E1 10273.375,E2 10273.375} C_VEL
LIN {X 0,Y 351.534,Z 569.588,A -85,B 0,C 180,E1 10270.737,E2 10270.737} C_VEL
LIN {X 0,Y 350.149,Z 567.05,A -85,B 0,C 180,E1 10269.201,E2 10269.201} C_VEL
LIN {X 0,Y 348.409,Z 563.632,A -85,B 0,C 180,E1 10266.757,E2 10266.757} C_VEL
LIN {X 0,Y 346.683,Z 559.566,A -85,B 0,C 180,E1 10262.479,E2 10262.479} C_VEL
LIN {X 0,Y 346.469,Z 559.255,A -85,B 0,C 180,E1 10258.015,E2 10258.015} C_VEL
LIN {X 0,Y 346.696,Z 559.676,A -85,B 0,C 180,E1 10256.859,E2 10256.859} C_VEL
LIN {X 0,Y 348.892,Z 564.484,A -85,B 0,C 180,E1 10251.927,E2 10251.927} C_VEL
LIN {X 0,Y 351.241,Z 568.975,A -85,B 0,C 180,E1 10249.005,E2 10249.005} C_VEL
LIN {X 0,Y 353.759,Z 573.797,A -85,B 0,C 180,E1 10246.599,E2 10246.599} C_VEL
LIN {X 0,Y 354.285,Z 575.067,A -85,B 0,C 180,E1 10246.13,E2 10246.13} C_VEL
LIN {X 0,Y 339.762,Z 721.588,A -85,B 0,C 180,E1 10243.419,E2 10243.419} C_VEL
LIN {X 0,Y 335.835,Z 745.18,A -85,B 0,C 180,E1 10242.857,E2 10242.857} C_VEL
LIN {X 0,Y 331.12,Z 766.11,A -85,B 0,C 180,E1 10242.195,E2 10242.195} C_VEL
LIN {X 0,Y 325.026,Z 787.16,A -85,B 0,C 180,E1 10241.327,E2 10241.327} C_VEL
LIN {X 0,Y 317.659,Z 808.401,A -85,B 0,C 180,E1 10240.222,E2 10240.222} C_VEL
LIN {X 0,Y 309.184,Z 828.721,A -85,B 0,C 180,E1 10238.884,E2 10238.884} C_VEL
LIN {X 0,Y 299.718,Z 848.635,A -85,B 0,C 180,E1 10237.263,E2 10237.263} C_VEL
LIN {X 0,Y 289.333,Z 867.55,A -85,B 0,C 180,E1 10235.333,E2 10235.333} C_VEL
LIN {X 0,Y 277.831,Z 886.342,A -85,B 0,C 180,E1 10232.947,E2 10232.947} C_VEL
LIN {X 0,Y 267.164,Z 902.063,A -85,B 0,C 180,E1 10230.461,E2 10230.461} C_VEL
LIN {X 0,Y 255.215,Z 918.205,A -85,B 0,C 180,E1 10227.272,E2 10227.272} C_VEL
LIN {X 0,Y 244.347,Z 931.86,A -85,B 0,C 180,E1 10223.896,E2 10223.896} C_VEL
LIN {X 0,Y 233.117,Z 945.073,A -85,B 0,C 180,E1 10219.761,E2 10219.761} C_VEL
LIN {X 0,Y 222.867,Z 956.753,A -85,B 0,C 180,E1 10215.133,E2 10215.133} C_VEL
LIN {X 0,Y 213.504,Z 967.039,A -85,B 0,C 180,E1 10209.822,E2 10209.822} C_VEL
LIN {X 0,Y 205.7,Z 975.842,A -85,B 0,C 180,E1 10203.98,E2 10203.98} C_VEL
LIN {X 0,Y 199.942,Z 982.6,A -85,B 0,C 180,E1 10198.034,E2 10198.034} C_VEL
LIN {X 0,Y 195.636,Z 988.366,A -85,B 0,C 180,E1 10191.273,E2 10191.273} C_VEL
LIN {X 0,Y 193.345,Z 992.101,A -85,B 0,C 180,E1 10184.983,E2 10184.983} C_VEL
LIN {X 0,Y 192.289,Z 994.649,A -85,B 0,C 180,E1 10178.37,E2 10178.37} C_VEL
LIN {X 0,Y 192.053,Z 995.621,A -85,B 0,C 180,E1 10172.684,E2 10172.684} C_VEL
LIN {X 0,Y 192.055,Z 995.672,A -85,B 0,C 180,E1 10167.911,E2 10167.911} C_VEL
LIN {X 0,Y 192.205,Z 994.931,A -85,B 0,C 180,E1 10162.828,E2 10162.828} C_VEL
LIN {X 0,Y 192.921,Z 993.041,A -85,B 0,C 180,E1 10156.819,E2 10156.819} C_VEL
LIN {X 0,Y 194.924,Z 989.435,A -85,B 0,C 180,E1 10150.213,E2 10150.213} C_VEL
LIN {X 0,Y 198.622,Z 984.39,A -85,B 0,C 180,E1 10143.644,E2 10143.644} C_VEL
LIN {X 0,Y 204.097,Z 977.688,A -85,B 0,C 180,E1 10137.396,E2 10137.396} C_VEL
LIN {X 0,Y 211.554,Z 969.339,A -85,B 0,C 180,E1 10131.405,E2 10131.405} C_VEL
LIN {X 0,Y 220.398,Z 959.482,A -85,B 0,C 180,E1 10126.05,E2 10126.05} C_VEL
LIN {X 0,Y 231.379,Z 947.168,A -85,B 0,C 180,E1 10120.874,E2 10120.874} C_VEL
LIN {X 0,Y 242.14,Z 934.653,A -85,B 0,C 180,E1 10116.775,E2 10116.775} C_VEL
LIN {X 0,Y 253.304,Z 920.798,A -85,B 0,C 180,E1 10113.203,E2 10113.203} C_VEL
LIN {X 0,Y 264.635,Z 905.84,A -85,B 0,C 180,E1 10110.102,E2 10110.102} C_VEL
LIN {X 0,Y 275.909,Z 889.454,A -85,B 0,C 180,E1 10107.402,E2 10107.402} C_VEL
LIN {X 0,Y 286.962,Z 871.97,A -85,B 0,C 180,E1 10105.066,E2 10105.066} C_VEL
LIN {X 0,Y 297.17,Z 853.675,A -85,B 0,C 180,E1 10103.115,E2 10103.115} C_VEL
LIN {X 0,Y 306.693,Z 834.677,A -85,B 0,C 180,E1 10101.461,E2 10101.461} C_VEL
LIN {X 0,Y 315.111,Z 815.141,A -85,B 0,C 180,E1 10100.096,E2 10100.096} C_VEL
LIN {X 0,Y 322.867,Z 794.382,A -85,B 0,C 180,E1 10098.919,E2 10098.919} C_VEL
LIN {X 0,Y 329.055,Z 774.213,A -85,B 0,C 180,E1 10098.015,E2 10098.015} C_VEL
LIN {X 0,Y 334.784,Z 751.19,A -85,B 0,C 180,E1 10097.209,E2 10097.209} C_VEL
LIN {X 0,Y 338.836,Z 729.079,A -85,B 0,C 180,E1 10096.642,E2 10096.642} C_VEL
LIN {X 0,Y 342.429,Z 698.232,A -85,B 0,C 180,E1 10096.035,E2 10096.035} C_VEL
LIN {X 0,Y 347.482,Z 646.068,A -85,B 0,C 180,E1 10095.072,E2 10095.072} C_VEL
LIN {X 0,Y 347.965,Z 638.531,A -85,B 0,C 180,E1 10094.774,E2 10094.774} C_VEL
LIN {X 0,Y 348.407,Z 618.954,A -85,B 0,C 180,E1 10093.418,E2 10093.418} C_VEL
LIN {X 0,Y 348.886,Z 612.473,A -85,B 0,C 180,E1 10093.178,E2 10093.178} C_VEL
LIN {X 0,Y 352.081,Z 580.67,A -85,B 0,C 180,E1 10092.59,E2 10092.59} C_VEL
LIN {X 0,Y 349.232,Z 575.06,A -85,B 0,C 180,E1 10089.559,E2 10089.559} C_VEL
LIN {X 0,Y 347.429,Z 571.55,A -85,B 0,C 180,E1 10086.943,E2 10086.943} C_VEL
LIN {X 0,Y 345.77,Z 567.295,A -85,B 0,C 180,E1 10082.155,E2 10082.155} C_VEL
LIN {X 0,Y 345.848,Z 567.553,A -85,B 0,C 180,E1 10077.847,E2 10077.847} C_VEL
LIN {X 0,Y 347.421,Z 571.518,A -85,B 0,C 180,E1 10073.556,E2 10073.556} C_VEL
LIN {X 0,Y 349.835,Z 576.189,A -85,B 0,C 180,E1 10070.209,E2 10070.209} C_VEL
LIN {X 0,Y 352.201,Z 580.97,A -85,B 0,C 180,E1 10067.777,E2 10067.777} C_VEL
LIN {X 0,Y 337.268,Z 728.456,A -85,B 0,C 180,E1 10065.074,E2 10065.074} C_VEL
LIN {X 0,Y 333.188,Z 752.335,A -85,B 0,C 180,E1 10064.543,E2 10064.543} C_VEL
LIN {X 0,Y 328.06,Z 774.169,A -85,B 0,C 180,E1 10063.944,E2 10063.944} C_VEL
LIN {X 0,Y 321.689,Z 795.18,A -85,B 0,C 180,E1 10063.178,E2 10063.178} C_VEL
LIN {X 0,Y 313.995,Z 816.58,A -85,B 0,C 180,E1 10062.177,E2 10062.177} C_VEL
LIN {X 0,Y 305.05,Z 837.3,A -85,B 0,C 180,E1 10060.926,E2 10060.926} C_VEL
LIN {X 0,Y 294.872,Z 857.976,A -85,B 0,C 180,E1 10059.353,E2 10059.353} C_VEL
LIN {X 0,Y 284.445,Z 876.477,A -85,B 0,C 180,E1 10057.575,E2 10057.575} C_VEL
LIN {X 0,Y 272.056,Z 896.186,A -85,B 0,C 180,E1 10055.186,E2 10055.186} C_VEL
LIN {X 0,Y 260.564,Z 912.748,A -85,B 0,C 180,E1 10052.653,E2 10052.653} C_VEL
LIN {X 0,Y 248.167,Z 929.062,A -85,B 0,C 180,E1 10049.493,E2 10049.493} C_VEL
LIN {X 0,Y 236.456,Z 943.544,A -85,B 0,C 180,E1 10045.966,E2 10045.966} C_VEL
LIN {X 0,Y 225.044,Z 956.719,A -85,B 0,C 180,E1 10041.843,E2 10041.843} C_VEL
LIN {X 0,Y 214.38,Z 968.789,A -85,B 0,C 180,E1 10037.069,E2 10037.069} C_VEL
LIN {X 0,Y 204.785,Z 979.39,A -85,B 0,C 180,E1 10031.602,E2 10031.602} C_VEL
LIN {X 0,Y 196.372,Z 989.054,A -85,B 0,C 180,E1 10025.121,E2 10025.121} C_VEL
LIN {X 0,Y 190.681,Z 996.162,A -85,B 0,C 180,E1 10018.84,E2 10018.84} C_VEL
LIN {X 0,Y 186.601,Z 1002.167,A -85,B 0,C 180,E1 10011.697,E2 10011.697} C_VEL
LIN {X 0,Y 184.732,Z 1005.984,A -85,B 0,C 180,E1 10005.379,E2 10005.379} C_VEL
LIN {X 0,Y 184.051,Z 1008.695,A -85,B 0,C 180,E1 9998.434,E2 9998.434} C_VEL
LIN {X 0,Y 184.016,Z 1009.689,A -85,B 0,C 180,E1 9993.115,E2 9993.115} C_VEL
LIN {X 0,Y 184.042,Z 1009.785,A -85,B 0,C 180,E1 9988.133,E2 9988.133} C_VEL
LIN {X 0,Y 184.007,Z 1009.052,A -85,B 0,C 180,E1 9983.136,E2 9983.136} C_VEL
LIN {X 0,Y 184.288,Z 1007.298,A -85,B 0,C 180,E1 9977.575,E2 9977.575} C_VEL
LIN {X 0,Y 185.797,Z 1003.658,A -85,B 0,C 180,E1 9970.513,E2 9970.513} C_VEL
LIN {X 0,Y 188.633,Z 998.949,A -85,B 0,C 180,E1 9964.241,E2 9964.241} C_VEL
LIN {X 0,Y 193.689,Z 992.296,A -85,B 0,C 180,E1 9957.535,E2 9957.535} C_VEL
LIN {X 0,Y 200.471,Z 984.211,A -85,B 0,C 180,E1 9951.438,E2 9951.438} C_VEL
LIN {X 0,Y 209.582,Z 974.005,A -85,B 0,C 180,E1 9945.476,E2 9945.476} C_VEL
LIN {X 0,Y 219.518,Z 962.902,A -85,B 0,C 180,E1 9940.487,E2 9940.487} C_VEL
LIN {X 0,Y 231.497,Z 949.192,A -85,B 0,C 180,E1 9935.72,E2 9935.72} C_VEL
LIN {X 0,Y 243.543,Z 934.817,A -85,B 0,C 180,E1 9931.818,E2 9931.818} C_VEL
LIN {X 0,Y 255.882,Z 918.871,A -85,B 0,C 180,E1 9928.469,E2 9928.469} C_VEL
LIN {X 0,Y 268.28,Z 901.637,A -85,B 0,C 180,E1 9925.604,E2 9925.604} C_VEL
LIN {X 0,Y 278.949,Z 885.28,A -85,B 0,C 180,E1 9923.439,E2 9923.439} C_VEL
LIN {X 0,Y 290.813,Z 865.148,A -85,B 0,C 180,E1 9921.311,E2 9921.311} C_VEL
LIN {X 0,Y 300.173,Z 847.252,A -85,B 0,C 180,E1 9919.801,E2 9919.801} C_VEL
LIN {X 0,Y 309.745,Z 826.401,A -85,B 0,C 180,E1 9918.393,E2 9918.393} C_VEL
LIN {X 0,Y 317.714,Z 806.216,A -85,B 0,C 180,E1 9917.315,E2 9917.315} C_VEL
LIN {X 0,Y 325.117,Z 783.705,A -85,B 0,C 180,E1 9916.383,E2 9916.383} C_VEL
LIN {X 0,Y 331.184,Z 761.034,A -85,B 0,C 180,E1 9915.68,E2 9915.68} C_VEL
LIN {X 0,Y 335.705,Z 737.687,A -85,B 0,C 180,E1 9915.128,E2 9915.128} C_VEL
LIN {X 0,Y 339.026,Z 711.385,A -85,B 0,C 180,E1 9914.606,E2 9914.606} C_VEL
LIN {X 0,Y 352.02,Z 580.793,A -85,B 0,C 180,E1 9912.216,E2 9912.216} C_VEL
LIN {X 0,Y 349.235,Z 575.28,A -85,B 0,C 180,E1 9909.309,E2 9909.309} C_VEL
LIN {X 0,Y 347.327,Z 571.51,A -85,B 0,C 180,E1 9906.612,E2 9906.612} C_VEL
LIN {X 0,Y 345.609,Z 567.241,A -85,B 0,C 180,E1 9901.989,E2 9901.989} C_VEL
LIN {X 0,Y 345.657,Z 567.381,A -85,B 0,C 180,E1 9897.181,E2 9897.181} C_VEL
LIN {X 0,Y 347.741,Z 572.306,A -85,B 0,C 180,E1 9892.15,E2 9892.15} C_VEL
LIN {X 0,Y 349.946,Z 576.676,A -85,B 0,C 180,E1 9889.297,E2 9889.297} C_VEL
LIN {X 0,Y 351.917,Z 580.67,A -85,B 0,C 180,E1 9887.298,E2 9887.298} C_VEL
LIN {X 0,Y 337.566,Z 721.919,A -85,B 0,C 180,E1 9884.72,E2 9884.72} C_VEL
LIN {X 0,Y 333.548,Z 745.564,A -85,B 0,C 180,E1 9884.17,E2 9884.17} C_VEL
LIN {X 0,Y 328.704,Z 766.638,A -85,B 0,C 180,E1 9883.518,E2 9883.518} C_VEL
LIN {X 0,Y 322.543,Z 787.47,A -85,B 0,C 180,E1 9882.68,E2 9882.68} C_VEL
LIN {X 0,Y 315.023,Z 808.711,A -85,B 0,C 180,E1 9881.601,E2 9881.601} C_VEL
LIN {X 0,Y 306.366,Z 829.03,A -85,B 0,C 180,E1 9880.294,E2 9880.294} C_VEL
LIN {X 0,Y 296.788,Z 848.744,A -85,B 0,C 180,E1 9878.725,E2 9878.725} C_VEL
LIN {X 0,Y 286.033,Z 867.859,A -85,B 0,C 180,E1 9876.813,E2 9876.813} C_VEL
LIN {X 0,Y 274.213,Z 886.652,A -85,B 0,C 180,E1 9874.467,E2 9874.467} C_VEL
LIN {X 0,Y 263.143,Z 902.478,A -85,B 0,C 180,E1 9871.996,E2 9871.996} C_VEL
LIN {X 0,Y 250.425,Z 919.057,A -85,B 0,C 180,E1 9868.731,E2 9868.731} C_VEL
LIN {X 0,Y 238.66,Z 933.288,A -85,B 0,C 180,E1 9865.188,E2 9865.188} C_VEL
LIN {X 0,Y 227.296,Z 946.007,A -85,B 0,C 180,E1 9861.124,E2 9861.124} C_VEL
LIN {X 0,Y 216.605,Z 957.598,A -85,B 0,C 180,E1 9856.438,E2 9856.438} C_VEL
LIN {X 0,Y 206.839,Z 967.748,A -85,B 0,C 180,E1 9851.052,E2 9851.052} C_VEL
LIN {X 0,Y 198.13,Z 976.941,A -85,B 0,C 180,E1 9844.656,E2 9844.656} C_VEL
LIN {X 0,Y 192.046,Z 983.706,A -85,B 0,C 180,E1 9838.372,E2 9838.372} C_VEL
LIN {X 0,Y 187.572,Z 989.267,A -85,B 0,C 180,E1 9831.249,E2 9831.249} C_VEL
LIN {X 0,Y 185.268,Z 992.864,A -85,B 0,C 180,E1 9824.691,E2 9824.691} C_VEL
LIN {X 0,Y 184.27,Z 995.078,A -85,B 0,C 180,E1 9818.108,E2 9818.108} C_VEL
LIN {X 0,Y 184.059,Z 995.922,A -85,B 0,C 180,E1 9812.801,E2 9812.801} C_VEL
LIN {X 0,Y 184.06,Z 995.972,A -85,B 0,C 180,E1 9807.82,E2 9807.82} C_VEL
LIN {X 0,Y 184.225,Z 995.232,A -85,B 0,C 180,E1 9802.516,E2 9802.516} C_VEL
LIN {X 0,Y 185.034,Z 993.344,A -85,B 0,C 180,E1 9796.246,E2 9796.246} C_VEL
LIN {X 0,Y 187.251,Z 989.741,A -85,B 0,C 180,E1 9789.366,E2 9789.366} C_VEL
LIN {X 0,Y 191.234,Z 984.746,A -85,B 0,C 180,E1 9782.609,E2 9782.609} C_VEL
LIN {X 0,Y 197.181,Z 977.997,A -85,B 0,C 180,E1 9776.101,E2 9776.101} C_VEL
LIN {X 0,Y 205.263,Z 969.521,A -85,B 0,C 180,E1 9769.887,E2 9769.887} C_VEL
LIN {X 0,Y 214.516,Z 959.79,A -85,B 0,C 180,E1 9764.515,E2 9764.515} C_VEL
LIN {X 0,Y 226.316,Z 947.183,A -85,B 0,C 180,E1 9759.181,E2 9759.181} C_VEL
LIN {X 0,Y 237.919,Z 934.272,A -85,B 0,C 180,E1 9754.974,E2 9754.974} C_VEL
LIN {X 0,Y 249.846,Z 919.919,A -85,B 0,C 180,E1 9751.349,E2 9751.349} C_VEL
LIN {X 0,Y 262.034,Z 904.219,A -85,B 0,C 180,E1 9748.195,E2 9748.195} C_VEL
LIN {X 0,Y 273.347,Z 888.125,A -85,B 0,C 180,E1 9745.636,E2 9745.636} C_VEL
LIN {X 0,Y 285.529,Z 868.971,A -85,B 0,C 180,E1 9743.203,E2 9743.203} C_VEL
LIN {X 0,Y 295.764,Z 850.891,A -85,B 0,C 180,E1 9741.368,E2 9741.368} C_VEL
LIN {X 0,Y 305.848,Z 830.509,A -85,B 0,C 180,E1 9739.71,E2 9739.71} C_VEL
LIN {X 0,Y 314.503,Z 810.448,A -85,B 0,C 180,E1 9738.399,E2 9738.399} C_VEL
LIN {X 0,Y 322.142,Z 789.195,A -85,B 0,C 180,E1 9737.299,E2 9737.299} C_VEL
LIN {X 0,Y 328.609,Z 767.72,A -85,B 0,C 180,E1 9736.42,E2 9736.42} C_VEL
LIN {X 0,Y 333.625,Z 746.024,A -85,B 0,C 180,E1 9735.744,E2 9735.744} C_VEL
LIN {X 0,Y 337.647,Z 722.678,A -85,B 0,C 180,E1 9735.196,E2 9735.196} C_VEL
LIN {X 0,Y 347.58,Z 625.438,A -85,B 0,C 180,E1 9733.411,E2 9733.411} C_VEL
LIN {X 0,Y 348.886,Z 612.473,A -85,B 0,C 180,E1 9733.178,E2 9733.178} C_VEL
LIN {X 0,Y 349.163,Z 607.477,A -85,B 0,C 180,E1 9732.923,E2 9732.923} C_VEL
LIN {X 0,Y 349.126,Z 595.074,A -85,B 0,C 180,E1 9731.7,E2 9731.7} C_VEL
LIN {X 0,Y 349.423,Z 590.761,A -85,B 0,C 180,E1 9731.502,E2 9731.502} C_VEL
LIN {X 0,Y 349.837,Z 586.486,A -85,B 0,C 180,E1 9731.401,E2 9731.401} C_VEL
LIN {X 0,Y 347.852,Z 582.541,A -85,B 0,C 180,E1 9729.096,E2 9729.096} C_VEL
LIN {X 0,Y 346.353,Z 579.429,A -85,B 0,C 180,E1 9726.798,E2 9726.798} C_VEL
LIN {X 0,Y 344.765,Z 575.224,A -85,B 0,C 180,E1 9721.995,E2 9721.995} C_VEL
LIN {X 0,Y 344.839,Z 575.444,A -85,B 0,C 180,E1 9718.006,E2 9718.006} C_VEL
LIN {X 0,Y 346.445,Z 579.521,A -85,B 0,C 180,E1 9713.538,E2 9713.538} C_VEL
LIN {X 0,Y 348.896,Z 584.668,A -85,B 0,C 180,E1 9710.099,E2 9710.099} C_VEL
LIN {X 0,Y 349.941,Z 586.956,A -85,B 0,C 180,E1 9708.947,E2 9708.947} C_VEL
LIN {X 0,Y 335.276,Z 728.251,A -85,B 0,C 180,E1 9706.402,E2 9706.402} C_VEL
LIN {X 0,Y 331.133,Z 752.052,A -85,B 0,C 180,E1 9705.885,E2 9705.885} C_VEL
LIN {X 0,Y 325.844,Z 774.187,A -85,B 0,C 180,E1 9705.296,E2 9705.296} C_VEL
LIN {X 0,Y 319.441,Z 794.884,A -85,B 0,C 180,E1 9704.568,E2 9704.568} C_VEL
LIN {X 0,Y 311.597,Z 816.302,A -85,B 0,C 180,E1 9703.598,E2 9703.598} C_VEL
LIN {X 0,Y 302.431,Z 837.11,A -85,B 0,C 180,E1 9702.379,E2 9702.379} C_VEL
LIN {X 0,Y 292.084,Z 857.673,A -85,B 0,C 180,E1 9700.856,E2 9700.856} C_VEL
LIN {X 0,Y 281.409,Z 876.172,A -85,B 0,C 180,E1 9699.124,E2 9699.124} C_VEL
LIN {X 0,Y 268.511,Z 896.137,A -85,B 0,C 180,E1 9696.753,E2 9696.753} C_VEL
LIN {X 0,Y 256.483,Z 912.953,A -85,B 0,C 180,E1 9694.214,E2 9694.214} C_VEL
LIN {X 0,Y 244.136,Z 928.636,A -85,B 0,C 180,E1 9691.205,E2 9691.205} C_VEL
LIN {X 0,Y 231.882,Z 943.233,A -85,B 0,C 180,E1 9687.678,E2 9687.678} C_VEL
LIN {X 0,Y 219.367,Z 957.054,A -85,B 0,C 180,E1 9683.333,E2 9683.333} C_VEL
LIN {X 0,Y 207.707,Z 969.53,A -85,B 0,C 180,E1 9678.251,E2 9678.251} C_VEL
LIN {X 0,Y 198.146,Z 979.548,A -85,B 0,C 180,E1 9672.934,E2 9672.934} C_VEL
LIN {X 0,Y 189.245,Z 989.106,A -85,B 0,C 180,E1 9666.277,E2 9666.277} C_VEL
LIN {X 0,Y 183.183,Z 996.164,A -85,B 0,C 180,E1 9659.779,E2 9659.779} C_VEL
LIN {X 0,Y 178.811,Z 1002.074,A -85,B 0,C 180,E1 9652.347,E2 9652.347} C_VEL
LIN {X 0,Y 176.788,Z 1005.845,A -85,B 0,C 180,E1 9645.751,E2 9645.751} C_VEL
LIN {X 0,Y 176.057,Z 1008.466,A -85,B 0,C 180,E1 9638.491,E2 9638.491} C_VEL
LIN {X 0,Y 176.024,Z 1009.413,A -85,B 0,C 180,E1 9632.931,E2 9632.931} C_VEL
LIN {X 0,Y 176.045,Z 1009.485,A -85,B 0,C 180,E1 9628.048,E2 9628.048} C_VEL
LIN {X 0,Y 176.009,Z 1008.75,A -85,B 0,C 180,E1 9622.822,E2 9622.822} C_VEL
LIN {X 0,Y 176.322,Z 1007.073,A -85,B 0,C 180,E1 9617.226,E2 9617.226} C_VEL
LIN {X 0,Y 177.937,Z 1003.564,A -85,B 0,C 180,E1 9609.958,E2 9609.958} C_VEL
LIN {X 0,Y 181.185,Z 998.637,A -85,B 0,C 180,E1 9603.099,E2 9603.099} C_VEL
LIN {X 0,Y 186.791,Z 991.87,A -85,B 0,C 180,E1 9596.065,E2 9596.065} C_VEL
LIN {X 0,Y 193.987,Z 983.895,A -85,B 0,C 180,E1 9589.895,E2 9589.895} C_VEL
LIN {X 0,Y 203.735,Z 973.622,A -85,B 0,C 180,E1 9583.786,E2 9583.786} C_VEL
LIN {X 0,Y 214.168,Z 962.585,A -85,B 0,C 180,E1 9578.781,E2 9578.781} C_VEL
LIN {X 0,Y 226.708,Z 948.875,A -85,B 0,C 180,E1 9574,E2 9574} C_VEL
LIN {X 0,Y 239.399,Z 934.323,A -85,B 0,C 180,E1 9570.078,E2 9570.078} C_VEL
LIN {X 0,Y 252.027,Z 918.557,A -85,B 0,C 180,E1 9566.808,E2 9566.808} C_VEL
LIN {X 0,Y 264.808,Z 901.323,A -85,B 0,C 180,E1 9563.989,E2 9563.989} C_VEL
LIN {X 0,Y 275.775,Z 884.967,A -85,B 0,C 180,E1 9561.868,E2 9561.868} C_VEL
LIN {X 0,Y 287.934,Z 864.836,A -85,B 0,C 180,E1 9559.791,E2 9559.791} C_VEL
LIN {X 0,Y 297.501,Z 846.952,A -85,B 0,C 180,E1 9558.323,E2 9558.323} C_VEL
LIN {X 0,Y 307.277,Z 826.09,A -85,B 0,C 180,E1 9556.955,E2 9556.955} C_VEL
LIN {X 0,Y 315.051,Z 806.808,A -85,B 0,C 180,E1 9555.952,E2 9555.952} C_VEL
LIN {X 0,Y 322.713,Z 784.136,A -85,B 0,C 180,E1 9555.034,E2 9555.034} C_VEL
LIN {X 0,Y 328.716,Z 762.212,A -85,B 0,C 180,E1 9554.371,E2 9554.371} C_VEL
LIN {X 0,Y 333.478,Z 738.668,A -85,B 0,C 180,E1 9553.822,E2 9553.822} C_VEL
LIN {X 0,Y 336.74,Z 714.504,A -85,B 0,C 180,E1 9553.345,E2 9553.345} C_VEL
LIN {X 0,Y 349.776,Z 586.573,A -85,B 0,C 180,E1 9551.041,E2 9551.041} C_VEL
LIN {X 0,Y 347.709,Z 582.543,A -85,B 0,C 180,E1 9548.683,E2 9548.683} C_VEL
LIN {X 0,Y 346.147,Z 579.257,A -85,B 0,C 180,E1 9546.301,E2 9546.301} C_VEL
LIN {X 0,Y 344.598,Z 575.169,A -85,B 0,C 180,E1 9541.829,E2 9541.829} C_VEL
LIN {X 0,Y 344.646,Z 575.276,A -85,B 0,C 180,E1 9537.339,E2 9537.339} C_VEL
LIN {X 0,Y 346.643,Z 580.256,A -85,B 0,C 180,E1 9532.292,E2 9532.292} C_VEL
LIN {X 0,Y 348.66,Z 584.376,A -85,B 0,C 180,E1 9529.591,E2 9529.591} C_VEL
LIN {X 0,Y 349.66,Z 586.632,A -85,B 0,C 180,E1 9528.476,E2 9528.476} C_VEL
LIN {X 0,Y 335.546,Z 722.245,A -85,B 0,C 180,E1 9526.038,E2 9526.038} C_VEL
LIN {X 0,Y 331.469,Z 745.807,A -85,B 0,C 180,E1 9525.503,E2 9525.503} C_VEL
LIN {X 0,Y 326.519,Z 766.95,A -85,B 0,C 180,E1 9524.868,E2 9524.868} C_VEL
LIN {X 0,Y 319.857,Z 788.929,A -85,B 0,C 180,E1 9524.001,E2 9524.001} C_VEL
LIN {X 0,Y 312.153,Z 810.109,A -85,B 0,C 180,E1 9522.942,E2 9522.942} C_VEL
LIN {X 0,Y 303.32,Z 830.231,A -85,B 0,C 180,E1 9521.666,E2 9521.666} C_VEL
LIN {X 0,Y 293.422,Z 849.979,A -85,B 0,C 180,E1 9520.114,E2 9520.114} C_VEL
LIN {X 0,Y 282.93,Z 868.168,A -85,B 0,C 180,E1 9518.327,E2 9518.327} C_VEL
LIN {X 0,Y 270.886,Z 886.831,A -85,B 0,C 180,E1 9516.045,E2 9516.045} C_VEL
LIN {X 0,Y 259.473,Z 902.684,A -85,B 0,C 180,E1 9513.612,E2 9513.612} C_VEL
LIN {X 0,Y 246.879,Z 918.626,A -85,B 0,C 180,E1 9510.533,E2 9510.533} C_VEL
LIN {X 0,Y 235.352,Z 932.086,A -85,B 0,C 180,E1 9507.253,E2 9507.253} C_VEL
LIN {X 0,Y 222.801,Z 945.696,A -85,B 0,C 180,E1 9503.006,E2 9503.006} C_VEL
LIN {X 0,Y 211.513,Z 957.378,A -85,B 0,C 180,E1 9498.314,E2 9498.314} C_VEL
LIN {X 0,Y 201.179,Z 967.559,A -85,B 0,C 180,E1 9492.906,E2 9492.906} C_VEL
LIN {X 0,Y 192.224,Z 976.464,A -85,B 0,C 180,E1 9486.733,E2 9486.733} C_VEL
LIN {X 0,Y 185.568,Z 983.22,A -85,B 0,C 180,E1 9480.425,E2 9480.425} C_VEL
LIN {X 0,Y 180.29,Z 989.18,A -85,B 0,C 180,E1 9472.839,E2 9472.839} C_VEL
LIN {X 0,Y 177.69,Z 992.712,A -85,B 0,C 180,E1 9466.338,E2 9466.338} C_VEL
LIN {X 0,Y 176.383,Z 995.253,A -85,B 0,C 180,E1 9459.131,E2 9459.131} C_VEL
LIN {X 0,Y 176.065,Z 996.222,A -85,B 0,C 180,E1 9452.928,E2 9452.928} C_VEL
LIN {X 0,Y 176.066,Z 996.272,A -85,B 0,C 180,E1 9447.721,E2 9447.721} C_VEL
LIN {X 0,Y 176.25,Z 995.534,A -85,B 0,C 180,E1 9442.175,E2 9442.175} C_VEL
LIN {X 0,Y 177.165,Z 993.648,A -85,B 0,C 180,E1 9435.623,E2 9435.623} C_VEL
LIN {X 0,Y 179.665,Z 989.982,A -85,B 0,C 180,E1 9428.339,E2 9428.339} C_VEL
LIN {X 0,Y 184.205,Z 984.795,A -85,B 0,C 180,E1 9421.115,E2 9421.115} C_VEL
LIN {X 0,Y 190.718,Z 977.964,A -85,B 0,C 180,E1 9414.417,E2 9414.417} C_VEL
LIN {X 0,Y 199.312,Z 969.51,A -85,B 0,C 180,E1 9408.153,E2 9408.153} C_VEL
LIN {X 0,Y 209.017,Z 959.883,A -85,B 0,C 180,E1 9402.788,E2 9402.788} C_VEL
LIN {X 0,Y 220.909,Z 947.784,A -85,B 0,C 180,E1 9397.628,E2 9397.628} C_VEL
LIN {X 0,Y 232.639,Z 935.267,A -85,B 0,C 180,E1 9393.518,E2 9393.518} C_VEL
LIN {X 0,Y 245.206,Z 920.775,A -85,B 0,C 180,E1 9389.833,E2 9389.833} C_VEL
LIN {X 0,Y 257.53,Z 905.52,A -85,B 0,C 180,E1 9386.762,E2 9386.762} C_VEL
LIN {X 0,Y 269.528,Z 888.976,A -85,B 0,C 180,E1 9384.15,E2 9384.15} C_VEL
LIN {X 0,Y 281.63,Z 870.594,A -85,B 0,C 180,E1 9381.829,E2 9381.829} C_VEL
LIN {X 0,Y 292.148,Z 852.54,A -85,B 0,C 180,E1 9380.014,E2 9380.014} C_VEL
LIN {X 0,Y 302.801,Z 831.7,A -85,B 0,C 180,E1 9378.335,E2 9378.335} C_VEL
LIN {X 0,Y 311.628,Z 811.742,A -85,B 0,C 180,E1 9377.053,E2 9377.053} C_VEL
LIN {X 0,Y 319.718,Z 789.862,A -85,B 0,C 180,E1 9375.941,E2 9375.941} C_VEL
LIN {X 0,Y 326.186,Z 768.904,A -85,B 0,C 180,E1 9375.102,E2 9375.102} C_VEL
LIN {X 0,Y 331.405,Z 746.96,A -85,B 0,C 180,E1 9374.429,E2 9374.429} C_VEL
LIN {X 0,Y 335.52,Z 723.917,A -85,B 0,C 180,E1 9373.896,E2 9373.896} C_VEL
LIN {X 0,Y 343.076,Z 652.384,A -85,B 0,C 180,E1 9372.596,E2 9372.596} C_VEL
LIN {X 0,Y 349.423,Z 590.761,A -85,B 0,C 180,E1 9371.502,E2 9371.502} C_VEL
LIN {X 0,Y 349.42,Z 588.796,A -85,B 0,C 180,E1 9371.294,E2 9371.294} C_VEL
LIN {X 0,Y 349.012,Z 587.534,A -85,B 0,C 180,E1 9370.809,E2 9370.809} C_VEL
LIN {X 0,Y 348.135,Z 587.41,A -85,B 0,C 180,E1 9369.99,E2 9369.99} C_VEL
LIN {X 0,Y 346.253,Z 588.966,A -85,B 0,C 180,E1 9368.202,E2 9368.202} C_VEL
LIN {X 0,Y 345.819,Z 588.568,A -85,B 0,C 180,E1 9367.607,E2 9367.607} C_VEL
LIN {X 0,Y 345.093,Z 587.051,A -85,B 0,C 180,E1 9366.321,E2 9366.321} C_VEL
LIN {X 0,Y 343.791,Z 583.165,A -85,B 0,C 180,E1 9362,E2 9362} C_VEL
LIN {X 0,Y 343.833,Z 583.335,A -85,B 0,C 180,E1 9358.167,E2 9358.167} C_VEL
LIN {X 0,Y 345.588,Z 588.009,A -85,B 0,C 180,E1 9353.271,E2 9353.271} C_VEL
LIN {X 0,Y 347.618,Z 592.363,A -85,B 0,C 180,E1 9350.397,E2 9350.397} C_VEL
LIN {X 0,Y 347.812,Z 593.038,A -85,B 0,C 180,E1 9350.137,E2 9350.137} C_VEL
LIN {X 0,Y 333.473,Z 727.996,A -85,B 0,C 180,E1 9347.745,E2 9347.745} C_VEL
LIN {X 0,Y 329.238,Z 751.879,A -85,B 0,C 180,E1 9347.241,E2 9347.241} C_VEL
LIN {X 0,Y 323.666,Z 774.707,A -85,B 0,C 180,E1 9346.651,E2 9346.651} C_VEL
LIN {X 0,Y 316.94,Z 795.878,A -85,B 0,C 180,E1 9345.924,E2 9345.924} C_VEL
LIN {X 0,Y 308.807,Z 817.406,A -85,B 0,C 180,E1 9344.968,E2 9344.968} C_VEL
LIN {X 0,Y 299.794,Z 837.378,A -85,B 0,C 180,E1 9343.827,E2 9343.827} C_VEL
LIN {X 0,Y 289.077,Z 858.111,A -85,B 0,C 180,E1 9342.326,E2 9342.326} C_VEL
LIN {X 0,Y 278.171,Z 876.542,A -85,B 0,C 180,E1 9340.636,E2 9340.636} C_VEL
LIN {X 0,Y 265.139,Z 896.135,A -85,B 0,C 180,E1 9338.352,E2 9338.352} C_VEL
LIN {X 0,Y 252.594,Z 913.165,A -85,B 0,C 180,E1 9335.823,E2 9335.823} C_VEL
LIN {X 0,Y 239.504,Z 929.184,A -85,B 0,C 180,E1 9332.763,E2 9332.763} C_VEL
LIN {X 0,Y 226.836,Z 943.673,A -85,B 0,C 180,E1 9329.25,E2 9329.25} C_VEL
LIN {X 0,Y 214.467,Z 956.742,A -85,B 0,C 180,E1 9325.129,E2 9325.129} C_VEL
LIN {X 0,Y 202.102,Z 969.324,A -85,B 0,C 180,E1 9319.974,E2 9319.974} C_VEL
LIN {X 0,Y 191.622,Z 979.706,A -85,B 0,C 180,E1 9314.357,E2 9314.357} C_VEL
LIN {X 0,Y 182.562,Z 988.793,A -85,B 0,C 180,E1 9307.832,E2 9307.832} C_VEL
LIN {X 0,Y 175.999,Z 995.853,A -85,B 0,C 180,E1 9301.127,E2 9301.127} C_VEL
LIN {X 0,Y 171.2,Z 1001.765,A -85,B 0,C 180,E1 9293.398,E2 9293.398} C_VEL
LIN {X 0,Y 168.915,Z 1005.55,A -85,B 0,C 180,E1 9286.482,E2 9286.482} C_VEL
LIN {X 0,Y 168.069,Z 1008.163,A -85,B 0,C 180,E1 9278.898,E2 9278.898} C_VEL
LIN {X 0,Y 168.027,Z 1009.113,A -85,B 0,C 180,E1 9273.071,E2 9273.071} C_VEL
LIN {X 0,Y 168.047,Z 1009.184,A -85,B 0,C 180,E1 9267.955,E2 9267.955} C_VEL
LIN {X 0,Y 168.017,Z 1008.447,A -85,B 0,C 180,E1 9262.479,E2 9262.479} C_VEL
LIN {X 0,Y 168.44,Z 1006.646,A -85,B 0,C 180,E1 9256.267,E2 9256.267} C_VEL
LIN {X 0,Y 170.465,Z 1002.822,A -85,B 0,C 180,E1 9248.317,E2 9248.317} C_VEL
LIN {X 0,Y 174.056,Z 998.046,A -85,B 0,C 180,E1 9241.509,E2 9241.509} C_VEL
LIN {X 0,Y 180.811,Z 990.573,A -85,B 0,C 180,E1 9233.729,E2 9233.729} C_VEL
LIN {X 0,Y 188.984,Z 982.287,A -85,B 0,C 180,E1 9227.341,E2 9227.341} C_VEL
LIN {X 0,Y 199.515,Z 971.789,A -85,B 0,C 180,E1 9221.269,E2 9221.269} C_VEL
LIN {X 0,Y 210.801,Z 960.51,A -85,B 0,C 180,E1 9216.271,E2 9216.271} C_VEL
LIN {X 0,Y 222.913,Z 947.715,A -85,B 0,C 180,E1 9211.956,E2 9211.956} C_VEL
LIN {X 0,Y 235.888,Z 933.347,A -85,B 0,C 180,E1 9208.172,E2 9208.172} C_VEL
LIN {X 0,Y 248.771,Z 917.773,A -85,B 0,C 180,E1 9205.013,E2 9205.013} C_VEL
LIN {X 0,Y 262.43,Z 899.759,A -85,B 0,C 180,E1 9202.159,E2 9202.159} C_VEL
LIN {X 0,Y 273.987,Z 882.893,A -85,B 0,C 180,E1 9200.061,E2 9200.061} C_VEL
LIN {X 0,Y 286.102,Z 863.041,A -85,B 0,C 180,E1 9198.111,E2 9198.111} C_VEL
LIN {X 0,Y 296.334,Z 844.178,A -85,B 0,C 180,E1 9196.64,E2 9196.64} C_VEL
LIN {X 0,Y 305.881,Z 823.757,A -85,B 0,C 180,E1 9195.384,E2 9195.384} C_VEL
LIN {X 0,Y 314.391,Z 802.75,A -85,B 0,C 180,E1 9194.362,E2 9194.362} C_VEL
LIN {X 0,Y 321.389,Z 781.597,A -85,B 0,C 180,E1 9193.57,E2 9193.57} C_VEL
LIN {X 0,Y 327.562,Z 758.828,A -85,B 0,C 180,E1 9192.928,E2 9192.928} C_VEL
LIN {X 0,Y 332.061,Z 735.911,A -85,B 0,C 180,E1 9192.421,E2 9192.421} C_VEL
LIN {X 0,Y 335.916,Z 705.022,A -85,B 0,C 180,E1 9191.841,E2 9191.841} C_VEL
LIN {X 0,Y 347.643,Z 592.671,A -85,B 0,C 180,E1 9189.853,E2 9189.853} C_VEL
LIN {X 0,Y 346.169,Z 589.671,A -85,B 0,C 180,E1 9187.969,E2 9187.969} C_VEL
LIN {X 0,Y 344.977,Z 587.001,A -85,B 0,C 180,E1 9185.989,E2 9185.989} C_VEL
LIN {X 0,Y 343.59,Z 583.095,A -85,B 0,C 180,E1 9181.667,E2 9181.667} C_VEL
LIN {X 0,Y 343.655,Z 583.357,A -85,B 0,C 180,E1 9177.331,E2 9177.331} C_VEL
LIN {X 0,Y 345.501,Z 588.072,A -85,B 0,C 180,E1 9172.517,E2 9172.517} C_VEL
LIN {X 0,Y 347.383,Z 592.075,A -85,B 0,C 180,E1 9169.888,E2 9169.888} C_VEL
LIN {X 0,Y 347.536,Z 592.755,A -85,B 0,C 180,E1 9169.664,E2 9169.664} C_VEL
LIN {X 0,Y 333.706,Z 722.566,A -85,B 0,C 180,E1 9167.371,E2 9167.371} C_VEL
LIN {X 0,Y 329.556,Z 746.121,A -85,B 0,C 180,E1 9166.85,E2 9166.85} C_VEL
LIN {X 0,Y 324.463,Z 767.478,A -85,B 0,C 180,E1 9166.228,E2 9166.228} C_VEL
LIN {X 0,Y 317.736,Z 789.238,A -85,B 0,C 180,E1 9165.394,E2 9165.394} C_VEL
LIN {X 0,Y 309.885,Z 810.417,A -85,B 0,C 180,E1 9164.366,E2 9164.366} C_VEL
LIN {X 0,Y 300.878,Z 830.54,A -85,B 0,C 180,E1 9163.126,E2 9163.126} C_VEL
LIN {X 0,Y 290.305,Z 851.089,A -85,B 0,C 180,E1 9161.546,E2 9161.546} C_VEL
LIN {X 0,Y 280.03,Z 868.477,A -85,B 0,C 180,E1 9159.873,E2 9159.873} C_VEL
LIN {X 0,Y 267.306,Z 887.653,A -85,B 0,C 180,E1 9157.571,E2 9157.571} C_VEL
LIN {X 0,Y 255.559,Z 903.495,A -85,B 0,C 180,E1 9155.171,E2 9155.171} C_VEL
LIN {X 0,Y 242.218,Z 919.769,A -85,B 0,C 180,E1 9152.039,E2 9152.039} C_VEL
LIN {X 0,Y 229.647,Z 933.912,A -85,B 0,C 180,E1 9148.567,E2 9148.567} C_VEL
LIN {X 0,Y 217.307,Z 946.631,A -85,B 0,C 180,E1 9144.518,E2 9144.518} C_VEL
LIN {X 0,Y 205.545,Z 958.223,A -85,B 0,C 180,E1 9139.784,E2 9139.784} C_VEL
LIN {X 0,Y 194.721,Z 968.317,A -85,B 0,C 180,E1 9134.286,E2 9134.286} C_VEL
LIN {X 0,Y 184.895,Z 977.459,A -85,B 0,C 180,E1 9127.661,E2 9127.661} C_VEL
LIN {X 0,Y 177.932,Z 984.116,A -85,B 0,C 180,E1 9121.125,E2 9121.125} C_VEL
LIN {X 0,Y 172.581,Z 989.685,A -85,B 0,C 180,E1 9113.559,E2 9113.559} C_VEL
LIN {X 0,Y 169.796,Z 993.17,A -85,B 0,C 180,E1 9106.768,E2 9106.768} C_VEL
LIN {X 0,Y 168.396,Z 995.619,A -85,B 0,C 180,E1 9099.223,E2 9099.223} C_VEL
LIN {X 0,Y 168.072,Z 996.522,A -85,B 0,C 180,E1 9093.068,E2 9093.068} C_VEL
LIN {X 0,Y 168.071,Z 996.572,A -85,B 0,C 180,E1 9087.613,E2 9087.613} C_VEL
LIN {X 0,Y 168.28,Z 995.835,A -85,B 0,C 180,E1 9081.802,E2 9081.802} C_VEL
LIN {X 0,Y 169.316,Z 993.952,A -85,B 0,C 180,E1 9074.941,E2 9074.941} C_VEL
LIN {X 0,Y 172.024,Z 990.354,A -85,B 0,C 180,E1 9067.444,E2 9067.444} C_VEL
LIN {X 0,Y 176.769,Z 985.362,A -85,B 0,C 180,E1 9060.151,E2 9060.151} C_VEL
LIN {X 0,Y 183.887,Z 978.433,A -85,B 0,C 180,E1 9053.063,E2 9053.063} C_VEL
LIN {X 0,Y 192.764,Z 970.266,A -85,B 0,C 180,E1 9046.795,E2 9046.795} C_VEL
LIN {X 0,Y 203.251,Z 960.408,A -85,B 0,C 180,E1 9041.185,E2 9041.185} C_VEL
LIN {X 0,Y 215.962,Z 948.092,A -85,B 0,C 180,E1 9035.891,E2 9035.891} C_VEL
LIN {X 0,Y 228.187,Z 935.574,A -85,B 0,C 180,E1 9031.791,E2 9031.791} C_VEL
LIN {X 0,Y 240.749,Z 921.627,A -85,B 0,C 180,E1 9028.259,E2 9028.259} C_VEL
LIN {X 0,Y 253.457,Z 906.427,A -85,B 0,C 180,E1 9025.217,E2 9025.217} C_VEL
LIN {X 0,Y 265.897,Z 889.827,A -85,B 0,C 180,E1 9022.622,E2 9022.622} C_VEL
LIN {X 0,Y 277.815,Z 872.349,A -85,B 0,C 180,E1 9020.433,E2 9020.433} C_VEL
LIN {X 0,Y 288.995,Z 853.673,A -85,B 0,C 180,E1 9018.58,E2 9018.58} C_VEL
LIN {X 0,Y 299.932,Z 832.89,A -85,B 0,C 180,E1 9016.933,E2 9016.933} C_VEL
LIN {X 0,Y 308.927,Z 813.036,A -85,B 0,C 180,E1 9015.683,E2 9015.683} C_VEL
LIN {X 0,Y 317.17,Z 791.431,A -85,B 0,C 180,E1 9014.603,E2 9014.603} C_VEL
LIN {X 0,Y 323.527,Z 771.404,A -85,B 0,C 180,E1 9013.812,E2 9013.812} C_VEL
LIN {X 0,Y 329.197,Z 748.675,A -85,B 0,C 180,E1 9013.117,E2 9013.117} C_VEL
LIN {X 0,Y 333.416,Z 726.075,A -85,B 0,C 180,E1 9012.599,E2 9012.599} C_VEL
LIN {X 0,Y 338.276,Z 682.79,A -85,B 0,C 180,E1 9011.816,E2 9011.816} C_VEL
LIN {X 0,Y 347.737,Z 592.614,A -85,B 0,C 180,E1 9010.228,E2 9010.228} C_VEL
LIN {X 0,Y 346.378,Z 589.794,A -85,B 0,C 180,E1 9008.466,E2 9008.466} C_VEL
LIN {X 0,Y 345.819,Z 588.568,A -85,B 0,C 180,E1 9007.607,E2 9007.607} C_VEL
LIN {X 0,Y 345.017,Z 587.778,A -85,B 0,C 180,E1 9006.342,E2 9006.342} C_VEL
LIN {X 0,Y 343.813,Z 589.109,A -85,B 0,C 180,E1 9004.421,E2 9004.421} C_VEL
LIN {X 0,Y 342.841,Z 591.05,A -85,B 0,C 180,E1 9002.098,E2 9002.098} C_VEL
LIN {X 0,Y 342.771,Z 591.087,A -85,B 0,C 180,E1 9001.722,E2 9001.722} C_VEL
LIN {X 0,Y 342.83,Z 591.226,A -85,B 0,C 180,E1 8998.329,E2 8998.329} C_VEL
LIN {X 0,Y 344.499,Z 595.953,A -85,B 0,C 180,E1 8993.417,E2 8993.417} C_VEL
LIN {X 0,Y 345.841,Z 599.066,A -85,B 0,C 180,E1 8991.341,E2 8991.341} C_VEL
LIN {X 0,Y 331.854,Z 727.745,A -85,B 0,C 180,E1 8989.102,E2 8989.102} C_VEL
LIN {X 0,Y 327.555,Z 751.59,A -85,B 0,C 180,E1 8988.614,E2 8988.614} C_VEL
LIN {X 0,Y 321.901,Z 774.414,A -85,B 0,C 180,E1 8988.048,E2 8988.048} C_VEL
LIN {X 0,Y 315.075,Z 795.568,A -85,B 0,C 180,E1 8987.352,E2 8987.352} C_VEL
LIN {X 0,Y 306.519,Z 817.744,A -85,B 0,C 180,E1 8986.401,E2 8986.401} C_VEL
LIN {X 0,Y 297.627,Z 837.078,A -85,B 0,C 180,E1 8985.333,E2 8985.333} C_VEL
LIN {X 0,Y 286.864,Z 857.526,A -85,B 0,C 180,E1 8983.907,E2 8983.907} C_VEL
LIN {X 0,Y 275.624,Z 876.128,A -85,B 0,C 180,E1 8982.259,E2 8982.259} C_VEL
LIN {X 0,Y 262.204,Z 895.828,A -85,B 0,C 180,E1 8980.031,E2 8980.031} C_VEL
LIN {X 0,Y 249.674,Z 912.38,A -85,B 0,C 180,E1 8977.64,E2 8977.64} C_VEL
LIN {X 0,Y 236.422,Z 928.168,A -85,B 0,C 180,E1 8974.714,E2 8974.714} C_VEL
LIN {X 0,Y 223.39,Z 942.611,A -85,B 0,C 180,E1 8971.304,E2 8971.304} C_VEL
LIN {X 0,Y 210.28,Z 955.943,A -85,B 0,C 180,E1 8967.177,E2 8967.177} C_VEL
LIN {X 0,Y 197.495,Z 968.376,A -85,B 0,C 180,E1 8962.158,E2 8962.158} C_VEL
LIN {X 0,Y 186.654,Z 978.495,A -85,B 0,C 180,E1 8956.713,E2 8956.713} C_VEL
LIN {X 0,Y 176.023,Z 988.48,A -85,B 0,C 180,E1 8949.504,E2 8949.504} C_VEL
LIN {X 0,Y 168.918,Z 995.541,A -85,B 0,C 180,E1 8942.589,E2 8942.589} C_VEL
LIN {X 0,Y 163.644,Z 1001.456,A -85,B 0,C 180,E1 8934.547,E2 8934.547} C_VEL
LIN {X 0,Y 160.996,Z 1005.4,A -85,B 0,C 180,E1 8926.97,E2 8926.97} C_VEL
LIN {X 0,Y 160.08,Z 1007.869,A -85,B 0,C 180,E1 8919.303,E2 8919.303} C_VEL
LIN {X 0,Y 160.028,Z 1008.788,A -85,B 0,C 180,E1 8913.583,E2 8913.583} C_VEL
LIN {X 0,Y 160.057,Z 1008.905,A -85,B 0,C 180,E1 8908.159,E2 8908.159} C_VEL
LIN {X 0,Y 160.021,Z 1008.218,A -85,B 0,C 180,E1 8902.462,E2 8902.462} C_VEL
LIN {X 0,Y 160.478,Z 1006.461,A -85,B 0,C 180,E1 8895.94,E2 8895.94} C_VEL
LIN {X 0,Y 162.533,Z 1002.944,A -85,B 0,C 180,E1 8887.964,E2 8887.964} C_VEL
LIN {X 0,Y 166.536,Z 998.012,A -85,B 0,C 180,E1 8880.512,E2 8880.512} C_VEL
LIN {X 0,Y 173.413,Z 990.988,A -85,B 0,C 180,E1 8872.748,E2 8872.748} C_VEL
LIN {X 0,Y 181.935,Z 982.847,A -85,B 0,C 180,E1 8866.183,E2 8866.183} C_VEL
LIN {X 0,Y 193.528,Z 972,A -85,B 0,C 180,E1 8859.673,E2 8859.673} C_VEL
LIN {X 0,Y 205.32,Z 960.78,A -85,B 0,C 180,E1 8854.626,E2 8854.626} C_VEL
LIN {X 0,Y 218.474,Z 947.529,A -85,B 0,C 180,E1 8850.134,E2 8850.134} C_VEL
LIN {X 0,Y 232.173,Z 932.911,A -85,B 0,C 180,E1 8846.331,E2 8846.331} C_VEL
LIN {X 0,Y 245.139,Z 917.741,A -85,B 0,C 180,E1 8843.305,E2 8843.305} C_VEL
LIN {X 0,Y 258.79,Z 900.32,A -85,B 0,C 180,E1 8840.584,E2 8840.584} C_VEL
LIN {X 0,Y 270.685,Z 883.439,A -85,B 0,C 180,E1 8838.521,E2 8838.521} C_VEL
LIN {X 0,Y 283.048,Z 863.786,A -85,B 0,C 180,E1 8836.626,E2 8836.626} C_VEL
LIN {X 0,Y 293.331,Z 845.3,A -85,B 0,C 180,E1 8835.216,E2 8835.216} C_VEL
LIN {X 0,Y 303.381,Z 824.457,A -85,B 0,C 180,E1 8833.959,E2 8833.959} C_VEL
LIN {X 0,Y 311.444,Z 805.051,A -85,B 0,C 180,E1 8833.034,E2 8833.034} C_VEL
LIN {X 0,Y 319.136,Z 782.77,A -85,B 0,C 180,E1 8832.21,E2 8832.21} C_VEL
LIN {X 0,Y 325.484,Z 760.118,A -85,B 0,C 180,E1 8831.586,E2 8831.586} C_VEL
LIN {X 0,Y 330.226,Z 736.734,A -85,B 0,C 180,E1 8831.08,E2 8831.08} C_VEL
LIN {X 0,Y 333.768,Z 710.276,A -85,B 0,C 180,E1 8830.588,E2 8830.588} C_VEL
LIN {X 0,Y 345.672,Z 598.68,A -85,B 0,C 180,E1 8828.65,E2 8828.65} C_VEL
LIN {X 0,Y 343.907,Z 594.879,A -85,B 0,C 180,E1 8825.84,E2 8825.84} C_VEL
LIN {X 0,Y 342.584,Z 591.022,A -85,B 0,C 180,E1 8821.505,E2 8821.505} C_VEL
LIN {X 0,Y 342.647,Z 591.249,A -85,B 0,C 180,E1 8817.491,E2 8817.491} C_VEL
LIN {X 0,Y 344.364,Z 595.887,A -85,B 0,C 180,E1 8812.744,E2 8812.744} C_VEL
LIN {X 0,Y 345.578,Z 598.733,A -85,B 0,C 180,E1 8810.87,E2 8810.87} C_VEL
LIN {X 0,Y 332.024,Z 723.081,A -85,B 0,C 180,E1 8808.714,E2 8808.714} C_VEL
LIN {X 0,Y 327.798,Z 746.569,A -85,B 0,C 180,E1 8808.21,E2 8808.21} C_VEL
LIN {X 0,Y 322.537,Z 768.222,A -85,B 0,C 180,E1 8807.597,E2 8807.597} C_VEL
LIN {X 0,Y 315.805,Z 789.548,A -85,B 0,C 180,E1 8806.806,E2 8806.806} C_VEL
LIN {X 0,Y 307.812,Z 810.726,A -85,B 0,C 180,E1 8805.81,E2 8805.81} C_VEL
LIN {X 0,Y 298.633,Z 830.849,A -85,B 0,C 180,E1 8804.609,E2 8804.609} C_VEL
LIN {X 0,Y 288.314,Z 850.597,A -85,B 0,C 180,E1 8803.144,E2 8803.144} C_VEL
LIN {X 0,Y 277.339,Z 868.786,A -85,B 0,C 180,E1 8801.45,E2 8801.45} C_VEL
LIN {X 0,Y 264.584,Z 887.581,A -85,B 0,C 180,E1 8799.257,E2 8799.257} C_VEL
LIN {X 0,Y 252.539,Z 903.412,A -85,B 0,C 180,E1 8796.923,E2 8796.923} C_VEL
LIN {X 0,Y 238.475,Z 920.08,A -85,B 0,C 180,E1 8793.783,E2 8793.783} C_VEL
LIN {X 0,Y 225.457,Z 934.223,A -85,B 0,C 180,E1 8790.355,E2 8790.355} C_VEL
LIN {X 0,Y 212.406,Z 947.147,A -85,B 0,C 180,E1 8786.257,E2 8786.257} C_VEL
LIN {X 0,Y 199.719,Z 959.037,A -85,B 0,C 180,E1 8781.342,E2 8781.342} C_VEL
LIN {X 0,Y 188.886,Z 968.629,A -85,B 0,C 180,E1 8776.039,E2 8776.039} C_VEL
LIN {X 0,Y 178.425,Z 977.77,A -85,B 0,C 180,E1 8769.282,E2 8769.282} C_VEL
LIN {X 0,Y 170.931,Z 984.426,A -85,B 0,C 180,E1 8762.553,E2 8762.553} C_VEL
LIN {X 0,Y 165.099,Z 989.994,A -85,B 0,C 180,E1 8754.696,E2 8754.696} C_VEL
LIN {X 0,Y 162.02,Z 993.476,A -85,B 0,C 180,E1 8747.598,E2 8747.598} C_VEL
LIN {X 0,Y 160.455,Z 995.921,A -85,B 0,C 180,E1 8739.684,E2 8739.684} C_VEL
LIN {X 0,Y 160.079,Z 996.822,A -85,B 0,C 180,E1 8733.221,E2 8733.221} C_VEL
LIN {X 0,Y 160.076,Z 996.893,A -85,B 0,C 180,E1 8727.851,E2 8727.851} C_VEL
LIN {X 0,Y 160.267,Z 996.264,A -85,B 0,C 180,E1 8722.111,E2 8722.111} C_VEL
LIN {X 0,Y 161.144,Z 994.684,A -85,B 0,C 180,E1 8715.63,E2 8715.63} C_VEL
LIN {X 0,Y 163.961,Z 991.254,A -85,B 0,C 180,E1 8707.409,E2 8707.409} C_VEL
LIN {X 0,Y 168.555,Z 986.647,A -85,B 0,C 180,E1 8700.116,E2 8700.116} C_VEL
LIN {X 0,Y 176.368,Z 979.608,A -85,B 0,C 180,E1 8692.25,E2 8692.25} C_VEL
LIN {X 0,Y 185.636,Z 971.593,A -85,B 0,C 180,E1 8685.755,E2 8685.755} C_VEL
LIN {X 0,Y 196.769,Z 961.722,A -85,B 0,C 180,E1 8679.896,E2 8679.896} C_VEL
LIN {X 0,Y 208.686,Z 950.886,A -85,B 0,C 180,E1 8674.994,E2 8674.994} C_VEL
LIN {X 0,Y 221.183,Z 938.632,A -85,B 0,C 180,E1 8670.817,E2 8670.817} C_VEL
LIN {X 0,Y 234.683,Z 924.518,A -85,B 0,C 180,E1 8667.083,E2 8667.083} C_VEL
LIN {X 0,Y 247.472,Z 909.797,A -85,B 0,C 180,E1 8664.075,E2 8664.075} C_VEL
LIN {X 0,Y 261.656,Z 891.774,A -85,B 0,C 180,E1 8661.205,E2 8661.205} C_VEL
LIN {X 0,Y 273.917,Z 874.402,A -85,B 0,C 180,E1 8659.037,E2 8659.037} C_VEL
LIN {X 0,Y 285.663,Z 855.428,A -85,B 0,C 180,E1 8657.17,E2 8657.17} C_VEL
LIN {X 0,Y 296.385,Z 835.868,A -85,B 0,C 180,E1 8655.627,E2 8655.627} C_VEL
LIN {X 0,Y 305.968,Z 815.329,A -85,B 0,C 180,E1 8654.346,E2 8654.346} C_VEL
LIN {X 0,Y 314.797,Z 793,A -85,B 0,C 180,E1 8653.244,E2 8653.244} C_VEL
LIN {X 0,Y 321.258,Z 773.169,A -85,B 0,C 180,E1 8652.476,E2 8652.476} C_VEL
LIN {X 0,Y 327.304,Z 749.741,A -85,B 0,C 180,E1 8651.772,E2 8651.772} C_VEL
LIN {X 0,Y 331.509,Z 727.816,A -85,B 0,C 180,E1 8651.279,E2 8651.279} C_VEL
LIN {X 0,Y 335.634,Z 693.365,A -85,B 0,C 180,E1 8650.662,E2 8650.662} C_VEL
LIN {X 0,Y 345.787,Z 598.621,A -85,B 0,C 180,E1 8649.025,E2 8649.025} C_VEL
LIN {X 0,Y 344.116,Z 595.059,A -85,B 0,C 180,E1 8646.339,E2 8646.339} C_VEL
LIN {X 0,Y 342.771,Z 591.087,A -85,B 0,C 180,E1 8641.722,E2 8641.722} C_VEL
LIN {X 0,Y 342.547,Z 592.013,A -85,B 0,C 180,E1 8640.526,E2 8640.526} C_VEL
LIN {X 0,Y 342.198,Z 595.642,A -85,B 0,C 180,E1 8638.851,E2 8638.851} C_VEL
LIN {X 0,Y 342.128,Z 600.622,A -85,B 0,C 180,E1 8636.729,E2 8636.729} C_VEL
LIN {X 0,Y 342.31,Z 601.579,A -85,B 0,C 180,E1 8635.991,E2 8635.991} C_VEL
LIN {X 0,Y 343.329,Z 603.64,A -85,B 0,C 180,E1 8633.731,E2 8633.731} C_VEL
LIN {X 0,Y 343.971,Z 605.579,A -85,B 0,C 180,E1 8632.551,E2 8632.551} C_VEL
LIN {X 0,Y 330.418,Z 727.538,A -85,B 0,C 180,E1 8630.471,E2 8630.471} C_VEL
LIN {X 0,Y 326.061,Z 751.301,A -85,B 0,C 180,E1 8630,E2 8630} C_VEL
LIN {X 0,Y 320.329,Z 774.121,A -85,B 0,C 180,E1 8629.458,E2 8629.458} C_VEL
LIN {X 0,Y 313.352,Z 795.417,A -85,B 0,C 180,E1 8628.79,E2 8628.79} C_VEL
LIN {X 0,Y 304.61,Z 817.673,A -85,B 0,C 180,E1 8627.874,E2 8627.874} C_VEL
LIN {X 0,Y 295.221,Z 837.684,A -85,B 0,C 180,E1 8626.807,E2 8626.807} C_VEL
LIN {X 0,Y 283.652,Z 858.988,A -85,B 0,C 180,E1 8625.352,E2 8625.352} C_VEL
LIN {X 0,Y 272.341,Z 877.215,A -85,B 0,C 180,E1 8623.768,E2 8623.768} C_VEL
LIN {X 0,Y 259.079,Z 896.083,A -85,B 0,C 180,E1 8621.674,E2 8621.674} C_VEL
LIN {X 0,Y 245.863,Z 913.054,A -85,B 0,C 180,E1 8619.269,E2 8619.269} C_VEL
LIN {X 0,Y 232.253,Z 928.668,A -85,B 0,C 180,E1 8616.399,E2 8616.399} C_VEL
LIN {X 0,Y 218.033,Z 943.758,A -85,B 0,C 180,E1 8612.817,E2 8612.817} C_VEL
LIN {X 0,Y 204.674,Z 956.765,A -85,B 0,C 180,E1 8608.739,E2 8608.739} C_VEL
LIN {X 0,Y 190.647,Z 969.645,A -85,B 0,C 180,E1 8603.354,E2 8603.354} C_VEL
LIN {X 0,Y 178.831,Z 980.149,A -85,B 0,C 180,E1 8597.429,E2 8597.429} C_VEL
LIN {X 0,Y 168.812,Z 988.897,A -85,B 0,C 180,E1 8590.652,E2 8590.652} C_VEL
LIN {X 0,Y 160.935,Z 996.231,A -85,B 0,C 180,E1 8582.996,E2 8582.996} C_VEL
LIN {X 0,Y 155.775,Z 1001.579,A -85,B 0,C 180,E1 8575.062,E2 8575.062} C_VEL
LIN {X 0,Y 152.921,Z 1005.562,A -85,B 0,C 180,E1 8566.719,E2 8566.719} C_VEL
LIN {X 0,Y 152.078,Z 1007.704,A -85,B 0,C 180,E1 8559.079,E2 8559.079} C_VEL
LIN {X 0,Y 152.033,Z 1008.513,A -85,B 0,C 180,E1 8553.394,E2 8553.394} C_VEL
LIN {X 0,Y 152.061,Z 1008.606,A -85,B 0,C 180,E1 8548.084,E2 8548.084} C_VEL
LIN {X 0,Y 152.037,Z 1007.915,A -85,B 0,C 180,E1 8542.064,E2 8542.064} C_VEL
LIN {X 0,Y 152.579,Z 1006.155,A -85,B 0,C 180,E1 8535.196,E2 8535.196} C_VEL
LIN {X 0,Y 154.911,Z 1002.634,A -85,B 0,C 180,E1 8526.818,E2 8526.818} C_VEL
LIN {X 0,Y 159.346,Z 997.699,A -85,B 0,C 180,E1 8519.039,E2 8519.039} C_VEL
LIN {X 0,Y 166.824,Z 990.672,A -85,B 0,C 180,E1 8511.007,E2 8511.007} C_VEL
LIN {X 0,Y 175.972,Z 982.531,A -85,B 0,C 180,E1 8504.289,E2 8504.289} C_VEL
LIN {X 0,Y 188.281,Z 971.684,A -85,B 0,C 180,E1 8497.707,E2 8497.707} C_VEL
LIN {X 0,Y 200.672,Z 960.463,A -85,B 0,C 180,E1 8492.654,E2 8492.654} C_VEL
LIN {X 0,Y 214.399,Z 947.214,A -85,B 0,C 180,E1 8488.201,E2 8488.201} C_VEL
LIN {X 0,Y 228.49,Z 932.716,A -85,B 0,C 180,E1 8484.484,E2 8484.484} C_VEL
LIN {X 0,Y 241.812,Z 917.614,A -85,B 0,C 180,E1 8481.53,E2 8481.53} C_VEL
LIN {X 0,Y 255.721,Z 900.381,A -85,B 0,C 180,E1 8478.899,E2 8478.899} C_VEL
LIN {X 0,Y 267.938,Z 883.476,A -85,B 0,C 180,E1 8476.89,E2 8476.89} C_VEL
LIN {X 0,Y 280.997,Z 863.158,A -85,B 0,C 180,E1 8474.996,E2 8474.996} C_VEL
LIN {X 0,Y 291.631,Z 844.373,A -85,B 0,C 180,E1 8473.625,E2 8473.625} C_VEL
LIN {X 0,Y 301.72,Z 823.708,A -85,B 0,C 180,E1 8472.439,E2 8472.439} C_VEL
LIN {X 0,Y 310.207,Z 803.534,A -85,B 0,C 180,E1 8471.527,E2 8471.527} C_VEL
LIN {X 0,Y 317.76,Z 781.716,A -85,B 0,C 180,E1 8470.766,E2 8470.766} C_VEL
LIN {X 0,Y 324.167,Z 758.979,A -85,B 0,C 180,E1 8470.173,E2 8470.173} C_VEL
LIN {X 0,Y 328.888,Z 735.764,A -85,B 0,C 180,E1 8469.691,E2 8469.691} C_VEL
LIN {X 0,Y 332.749,Z 706.553,A -85,B 0,C 180,E1 8469.165,E2 8469.165} C_VEL
LIN {X 0,Y 343.785,Z 605.137,A -85,B 0,C 180,E1 8467.416,E2 8467.416} C_VEL
LIN {X 0,Y 342.753,Z 602.621,A -85,B 0,C 180,E1 8465.524,E2 8465.524} C_VEL
LIN {X 0,Y 341.581,Z 598.949,A -85,B 0,C 180,E1 8461.341,E2 8461.341} C_VEL
LIN {X 0,Y 341.641,Z 599.141,A -85,B 0,C 180,E1 8457.651,E2 8457.651} C_VEL
LIN {X 0,Y 343.233,Z 603.702,A -85,B 0,C 180,E1 8452.972,E2 8452.972} C_VEL
LIN {X 0,Y 343.716,Z 605.244,A -85,B 0,C 180,E1 8452.08,E2 8452.08} C_VEL
LIN {X 0,Y 330.55,Z 723.413,A -85,B 0,C 180,E1 8450.074,E2 8450.074} C_VEL
LIN {X 0,Y 326.25,Z 746.911,A -85,B 0,C 180,E1 8449.585,E2 8449.585} C_VEL
LIN {X 0,Y 320.826,Z 768.856,A -85,B 0,C 180,E1 8448.986,E2 8448.986} C_VEL
LIN {X 0,Y 313.887,Z 790.37,A -85,B 0,C 180,E1 8448.212,E2 8448.212} C_VEL
LIN {X 0,Y 305.489,Z 812.036,A -85,B 0,C 180,E1 8447.219,E2 8447.219} C_VEL
LIN {X 0,Y 296.15,Z 832.05,A -85,B 0,C 180,E1 8446.056,E2 8446.056} C_VEL
LIN {X 0,Y 284.84,Z 852.958,A -85,B 0,C 180,E1 8444.527,E2 8444.527} C_VEL
LIN {X 0,Y 273.641,Z 870.99,A -85,B 0,C 180,E1 8442.867,E2 8442.867} C_VEL
LIN {X 0,Y 260.56,Z 889.535,A -85,B 0,C 180,E1 8440.712,E2 8440.712} C_VEL
LIN {X 0,Y 247.527,Z 906.115,A -85,B 0,C 180,E1 8438.27,E2 8438.27} C_VEL
LIN {X 0,Y 234.193,Z 921.222,A -85,B 0,C 180,E1 8435.403,E2 8435.403} C_VEL
LIN {X 0,Y 220.772,Z 935.27,A -85,B 0,C 180,E1 8432.009,E2 8432.009} C_VEL
LIN {X 0,Y 207.402,Z 947.948,A -85,B 0,C 180,E1 8427.974,E2 8427.974} C_VEL
LIN {X 0,Y 194.049,Z 959.852,A -85,B 0,C 180,E1 8422.992,E2 8422.992} C_VEL
LIN {X 0,Y 182.706,Z 969.388,A -85,B 0,C 180,E1 8417.62,E2 8417.62} C_VEL
LIN {X 0,Y 171.67,Z 978.423,A -85,B 0,C 180,E1 8410.71,E2 8410.71} C_VEL
LIN {X 0,Y 163.388,Z 985.321,A -85,B 0,C 180,E1 8403.414,E2 8403.414} C_VEL
LIN {X 0,Y 157.469,Z 990.499,A -85,B 0,C 180,E1 8395.576,E2 8395.576} C_VEL
LIN {X 0,Y 154.154,Z 993.934,A -85,B 0,C 180,E1 8388.136,E2 8388.136} C_VEL
LIN {X 0,Y 152.471,Z 996.286,A -85,B 0,C 180,E1 8379.815,E2 8379.815} C_VEL
LIN {X 0,Y 152.088,Z 997.122,A -85,B 0,C 180,E1 8373.391,E2 8373.391} C_VEL
LIN {X 0,Y 152.082,Z 997.193,A -85,B 0,C 180,E1 8367.738,E2 8367.738} C_VEL
LIN {X 0,Y 152.299,Z 996.566,A -85,B 0,C 180,E1 8361.695,E2 8361.695} C_VEL
LIN {X 0,Y 153.303,Z 994.982,A -85,B 0,C 180,E1 8354.859,E2 8354.859} C_VEL
LIN {X 0,Y 156.431,Z 991.56,A -85,B 0,C 180,E1 8346.256,E2 8346.256} C_VEL
LIN {X 0,Y 161.465,Z 986.955,A -85,B 0,C 180,E1 8338.66,E2 8338.66} C_VEL
LIN {X 0,Y 169.91,Z 979.916,A -85,B 0,C 180,E1 8330.544,E2 8330.544} C_VEL
LIN {X 0,Y 179.517,Z 972.12,A -85,B 0,C 180,E1 8324.075,E2 8324.075} C_VEL
LIN {X 0,Y 191.447,Z 962.128,A -85,B 0,C 180,E1 8318.045,E2 8318.045} C_VEL
LIN {X 0,Y 204.058,Z 951.194,A -85,B 0,C 180,E1 8313.092,E2 8313.092} C_VEL
LIN {X 0,Y 217.233,Z 938.785,A -85,B 0,C 180,E1 8308.901,E2 8308.901} C_VEL
LIN {X 0,Y 231.052,Z 924.823,A -85,B 0,C 180,E1 8305.266,E2 8305.266} C_VEL
LIN {X 0,Y 244.24,Z 910.102,A -85,B 0,C 180,E1 8302.317,E2 8302.317} C_VEL
LIN {X 0,Y 258.813,Z 892.077,A -85,B 0,C 180,E1 8299.518,E2 8299.518} C_VEL
LIN {X 0,Y 271.371,Z 874.703,A -85,B 0,C 180,E1 8297.412,E2 8297.412} C_VEL
LIN {X 0,Y 283.375,Z 855.728,A -85,B 0,C 180,E1 8295.603,E2 8295.603} C_VEL
LIN {X 0,Y 294.414,Z 835.953,A -85,B 0,C 180,E1 8294.097,E2 8294.097} C_VEL
LIN {X 0,Y 304.154,Z 815.437,A -85,B 0,C 180,E1 8292.864,E2 8292.864} C_VEL
LIN {X 0,Y 313.247,Z 792.742,A -85,B 0,C 180,E1 8291.788,E2 8291.788} C_VEL
LIN {X 0,Y 319.848,Z 772.724,A -85,B 0,C 180,E1 8291.047,E2 8291.047} C_VEL
LIN {X 0,Y 325.879,Z 749.509,A -85,B 0,C 180,E1 8290.381,E2 8290.381} C_VEL
LIN {X 0,Y 330.181,Z 727.29,A -85,B 0,C 180,E1 8289.901,E2 8289.901} C_VEL
LIN {X 0,Y 334.74,Z 689.085,A -85,B 0,C 180,E1 8289.236,E2 8289.236} C_VEL
LIN {X 0,Y 343.931,Z 605.122,A -85,B 0,C 180,E1 8287.812,E2 8287.812} C_VEL
LIN {X 0,Y 342.963,Z 602.809,A -85,B 0,C 180,E1 8286.025,E2 8286.025} C_VEL
LIN {X 0,Y 341.789,Z 599.025,A -85,B 0,C 180,E1 8281.677,E2 8281.677} C_VEL
LIN {X 0,Y 341.839,Z 599.3,A -85,B 0,C 180,E1 8278.324,E2 8278.324} C_VEL
LIN {X 0,Y 342.31,Z 601.579,A -85,B 0,C 180,E1 8275.991,E2 8275.991} C_VEL
LIN {X 0,Y 342.45,Z 603.23,A -85,B 0,C 180,E1 8275.278,E2 8275.278} C_VEL
LIN {X 0,Y 342.379,Z 606.851,A -85,B 0,C 180,E1 8274.599,E2 8274.599} C_VEL
LIN {X 0,Y 342.055,Z 612.33,A -85,B 0,C 180,E1 8274.032,E2 8274.032} C_VEL
LIN {X 0,Y 341.433,Z 619.353,A -85,B 0,C 180,E1 8273.664,E2 8273.664} C_VEL
LIN {X 0,Y 341.258,Z 620.974,A -85,B 0,C 180,E1 8273.627,E2 8273.627} C_VEL
LIN {X 0,Y 329.151,Z 727.489,A -85,B 0,C 180,E1 8271.849,E2 8271.849} C_VEL
LIN {X 0,Y 324.731,Z 751.143,A -85,B 0,C 180,E1 8271.396,E2 8271.396} C_VEL
LIN {X 0,Y 318.953,Z 773.828,A -85,B 0,C 180,E1 8270.881,E2 8270.881} C_VEL
LIN {X 0,Y 311.927,Z 794.993,A -85,B 0,C 180,E1 8270.252,E2 8270.252} C_VEL
LIN {X 0,Y 303.113,Z 817.147,A -85,B 0,C 180,E1 8269.385,E2 8269.385} C_VEL
LIN {X 0,Y 293.469,Z 837.384,A -85,B 0,C 180,E1 8268.355,E2 8268.355} C_VEL
LIN {X 0,Y 281.856,Z 858.42,A -85,B 0,C 180,E1 8266.982,E2 8266.982} C_VEL
LIN {X 0,Y 270.558,Z 876.304,A -85,B 0,C 180,E1 8265.496,E2 8265.496} C_VEL
LIN {X 0,Y 257.165,Z 895.046,A -85,B 0,C 180,E1 8263.512,E2 8263.512} C_VEL
LIN {X 0,Y 243.885,Z 911.722,A -85,B 0,C 180,E1 8261.251,E2 8261.251} C_VEL
LIN {X 0,Y 229.944,Z 927.396,A -85,B 0,C 180,E1 8258.502,E2 8258.502} C_VEL
LIN {X 0,Y 215.859,Z 941.989,A -85,B 0,C 180,E1 8255.2,E2 8255.2} C_VEL
LIN {X 0,Y 201.866,Z 955.157,A -85,B 0,C 180,E1 8251.236,E2 8251.236} C_VEL
LIN {X 0,Y 188.311,Z 967.222,A -85,B 0,C 180,E1 8246.463,E2 8246.463} C_VEL
LIN {X 0,Y 175.621,Z 977.823,A -85,B 0,C 180,E1 8240.734,E2 8240.734} C_VEL
LIN {X 0,Y 163.534,Z 987.774,A -85,B 0,C 180,E1 8233.318,E2 8233.318} C_VEL
LIN {X 0,Y 155.107,Z 994.917,A -85,B 0,C 180,E1 8225.913,E2 8225.913} C_VEL
LIN {X 0,Y 148.729,Z 1000.835,A -85,B 0,C 180,E1 8217.201,E2 8217.201} C_VEL
LIN {X 0,Y 145.392,Z 1004.786,A -85,B 0,C 180,E1 8208.857,E2 8208.857} C_VEL
LIN {X 0,Y 144.12,Z 1007.253,A -85,B 0,C 180,E1 8200.392,E2 8200.392} C_VEL
LIN {X 0,Y 144.036,Z 1008.187,A -85,B 0,C 180,E1 8193.981,E2 8193.981} C_VEL
LIN {X 0,Y 144.069,Z 1008.332,A -85,B 0,C 180,E1 8188.411,E2 8188.411} C_VEL
LIN {X 0,Y 144.041,Z 1007.685,A -85,B 0,C 180,E1 8182.022,E2 8182.022} C_VEL
LIN {X 0,Y 144.633,Z 1005.97,A -85,B 0,C 180,E1 8174.773,E2 8174.773} C_VEL
LIN {X 0,Y 147.18,Z 1002.539,A -85,B 0,C 180,E1 8165.95,E2 8165.95} C_VEL
LIN {X 0,Y 152.262,Z 997.386,A -85,B 0,C 180,E1 8157.426,E2 8157.426} C_VEL
LIN {X 0,Y 160.402,Z 990.357,A -85,B 0,C 180,E1 8149.124,E2 8149.124} C_VEL
LIN {X 0,Y 170.213,Z 982.214,A -85,B 0,C 180,E1 8142.265,E2 8142.265} C_VEL
LIN {X 0,Y 183.264,Z 971.367,A -85,B 0,C 180,E1 8135.629,E2 8135.629} C_VEL
LIN {X 0,Y 196.275,Z 960.147,A -85,B 0,C 180,E1 8130.593,E2 8130.593} C_VEL
LIN {X 0,Y 210.579,Z 946.898,A -85,B 0,C 180,E1 8126.197,E2 8126.197} C_VEL
LIN {X 0,Y 225.162,Z 932.401,A -85,B 0,C 180,E1 8122.552,E2 8122.552} C_VEL
LIN {X 0,Y 239.3,Z 916.83,A -85,B 0,C 180,E1 8119.597,E2 8119.597} C_VEL
LIN {X 0,Y 254.016,Z 898.945,A -85,B 0,C 180,E1 8116.986,E2 8116.986} C_VEL
LIN {X 0,Y 266.582,Z 881.872,A -85,B 0,C 180,E1 8115.056,E2 8115.056} C_VEL
LIN {X 0,Y 279.436,Z 862.105,A -85,B 0,C 180,E1 8113.312,E2 8113.312} C_VEL
LIN {X 0,Y 290.726,Z 842.427,A -85,B 0,C 180,E1 8111.952,E2 8111.952} C_VEL
LIN {X 0,Y 300.944,Z 821.484,A -85,B 0,C 180,E1 8110.83,E2 8110.83} C_VEL
LIN {X 0,Y 309.593,Z 800.937,A -85,B 0,C 180,E1 8109.968,E2 8109.968} C_VEL
LIN {X 0,Y 316.823,Z 779.92,A -85,B 0,C 180,E1 8109.291,E2 8109.291} C_VEL
LIN {X 0,Y 323.261,Z 756.798,A -85,B 0,C 180,E1 8108.727,E2 8108.727} C_VEL
LIN {X 0,Y 327.804,Z 734.469,A -85,B 0,C 180,E1 8108.285,E2 8108.285} C_VEL
LIN {X 0,Y 331.871,Z 703.417,A -85,B 0,C 180,E1 8107.744,E2 8107.744} C_VEL
LIN {X 0,Y 342.093,Z 611.533,A -85,B 0,C 180,E1 8106.208,E2 8106.208} C_VEL
LIN {X 0,Y 341.385,Z 609.962,A -85,B 0,C 180,E1 8104.704,E2 8104.704} C_VEL
LIN {X 0,Y 340.581,Z 606.876,A -85,B 0,C 180,E1 8101.177,E2 8101.177} C_VEL
LIN {X 0,Y 340.639,Z 607.031,A -85,B 0,C 180,E1 8097.813,E2 8097.813} C_VEL
LIN {X 0,Y 342.053,Z 611.358,A -85,B 0,C 180,E1 8093.311,E2 8093.311} C_VEL
LIN {X 0,Y 329.264,Z 723.747,A -85,B 0,C 180,E1 8091.445,E2 8091.445} C_VEL
LIN {X 0,Y 324.907,Z 747.189,A -85,B 0,C 180,E1 8090.974,E2 8090.974} C_VEL
LIN {X 0,Y 319.391,Z 769.168,A -85,B 0,C 180,E1 8090.398,E2 8090.398} C_VEL
LIN {X 0,Y 312.303,Z 790.798,A -85,B 0,C 180,E1 8089.65,E2 8089.65} C_VEL
LIN {X 0,Y 303.809,Z 812.344,A -85,B 0,C 180,E1 8088.701,E2 8088.701} C_VEL
LIN {X 0,Y 294.309,Z 832.359,A -85,B 0,C 180,E1 8087.581,E2 8087.581} C_VEL
LIN {X 0,Y 283.151,Z 852.669,A -85,B 0,C 180,E1 8086.156,E2 8086.156} C_VEL
LIN {X 0,Y 271.735,Z 870.726,A -85,B 0,C 180,E1 8084.562,E2 8084.562} C_VEL
LIN {X 0,Y 258.407,Z 889.296,A -85,B 0,C 180,E1 8082.49,E2 8082.49} C_VEL
LIN {X 0,Y 245.438,Z 905.425,A -85,B 0,C 180,E1 8080.207,E2 8080.207} C_VEL
LIN {X 0,Y 231.538,Z 920.858,A -85,B 0,C 180,E1 8077.397,E2 8077.397} C_VEL
LIN {X 0,Y 217.776,Z 934.846,A -85,B 0,C 180,E1 8074.127,E2 8074.127} C_VEL
LIN {X 0,Y 203.925,Z 947.566,A -85,B 0,C 180,E1 8070.196,E2 8070.196} C_VEL
LIN {X 0,Y 190.292,Z 959.296,A -85,B 0,C 180,E1 8065.425,E2 8065.425} C_VEL
LIN {X 0,Y 177.79,Z 969.253,A -85,B 0,C 180,E1 8059.883,E2 8059.883} C_VEL
LIN {X 0,Y 165.949,Z 978.393,A -85,B 0,C 180,E1 8052.902,E2 8052.902} C_VEL
LIN {X 0,Y 157.275,Z 985.046,A -85,B 0,C 180,E1 8045.788,E2 8045.788} C_VEL
LIN {X 0,Y 150.355,Z 990.61,A -85,B 0,C 180,E1 8037.308,E2 8037.308} C_VEL
LIN {X 0,Y 146.566,Z 994.088,A -85,B 0,C 180,E1 8029.525,E2 8029.525} C_VEL
LIN {X 0,Y 144.576,Z 996.526,A -85,B 0,C 180,E1 8020.759,E2 8020.759} C_VEL
LIN {X 0,Y 144.097,Z 997.423,A -85,B 0,C 180,E1 8013.579,E2 8013.579} C_VEL
LIN {X 0,Y 144.087,Z 997.493,A -85,B 0,C 180,E1 8007.613,E2 8007.613} C_VEL
LIN {X 0,Y 144.341,Z 996.867,A -85,B 0,C 180,E1 8001.234,E2 8001.234} C_VEL
LIN {X 0,Y 145.48,Z 995.292,A -85,B 0,C 180,E1 7994.044,E2 7994.044} C_VEL
LIN {X 0,Y 148.974,Z 991.858,A -85,B 0,C 180,E1 7984.969,E2 7984.969} C_VEL
LIN {X 0,Y 154.489,Z 987.263,A -85,B 0,C 180,E1 7977.071,E2 7977.071} C_VEL
LIN {X 0,Y 163.614,Z 980.225,A -85,B 0,C 180,E1 7968.705,E2 7968.705} C_VEL
LIN {X 0,Y 173.861,Z 972.429,A -85,B 0,C 180,E1 7962.115,E2 7962.115} C_VEL
LIN {X 0,Y 185.96,Z 962.842,A -85,B 0,C 180,E1 7956.251,E2 7956.251} C_VEL
LIN {X 0,Y 198.98,Z 952.079,A -85,B 0,C 180,E1 7951.334,E2 7951.334} C_VEL
LIN {X 0,Y 212.821,Z 939.602,A -85,B 0,C 180,E1 7947.112,E2 7947.112} C_VEL
LIN {X 0,Y 226.884,Z 925.961,A -85,B 0,C 180,E1 7943.574,E2 7943.574} C_VEL
LIN {X 0,Y 240.43,Z 911.319,A -85,B 0,C 180,E1 7940.676,E2 7940.676} C_VEL
LIN {X 0,Y 254.565,Z 894.508,A -85,B 0,C 180,E1 7938.077,E2 7938.077} C_VEL
LIN {X 0,Y 267.314,Z 877.411,A -85,B 0,C 180,E1 7936.017,E2 7936.017} C_VEL
LIN {X 0,Y 280.419,Z 857.483,A -85,B 0,C 180,E1 7934.132,E2 7934.132} C_VEL
LIN {X 0,Y 291.643,Z 837.988,A -85,B 0,C 180,E1 7932.675,E2 7932.675} C_VEL
LIN {X 0,Y 301.622,Z 817.579,A -85,B 0,C 180,E1 7931.473,E2 7931.473} C_VEL
LIN {X 0,Y 310.138,Z 797.407,A -85,B 0,C 180,E1 7930.52,E2 7930.52} C_VEL
LIN {X 0,Y 317.069,Z 777.288,A -85,B 0,C 180,E1 7929.769,E2 7929.769} C_VEL
LIN {X 0,Y 323.345,Z 755.107,A -85,B 0,C 180,E1 7929.113,E2 7929.113} C_VEL
LIN {X 0,Y 328.059,Z 732.267,A -85,B 0,C 180,E1 7928.615,E2 7928.615} C_VEL
LIN {X 0,Y 331.803,Z 705.124,A -85,B 0,C 180,E1 7928.141,E2 7928.141} C_VEL
LIN {X 0,Y 342.247,Z 611.512,A -85,B 0,C 180,E1 7926.589,E2 7926.589} C_VEL
LIN {X 0,Y 340.792,Z 606.954,A -85,B 0,C 180,E1 7921.513,E2 7921.513} C_VEL
LIN {X 0,Y 340.839,Z 607.189,A -85,B 0,C 180,E1 7918.488,E2 7918.488} C_VEL
LIN {X 0,Y 342.248,Z 611.58,A -85,B 0,C 180,E1 7913.879,E2 7913.879} C_VEL
LIN {X 0,Y 342.259,Z 612.063,A -85,B 0,C 180,E1 7913.774,E2 7913.774} C_VEL
LIN {X 0,Y 341.258,Z 620.974,A -85,B 0,C 180,E1 7913.627,E2 7913.627} C_VEL
LIN {X 0,Y 340.283,Z 628.671,A -85,B 0,C 180,E1 7913.662,E2 7913.662} C_VEL
LIN {X 0,Y 337.275,Z 649.275,A -85,B 0,C 180,E1 7914.38,E2 7914.38} C_VEL
LIN {X 0,Y 336.443,Z 655.886,A -85,B 0,C 180,E1 7914.407,E2 7914.407} C_VEL
LIN {X 0,Y 327.961,Z 728.282,A -85,B 0,C 180,E1 7913.222,E2 7913.222} C_VEL
LIN {X 0,Y 323.429,Z 751.716,A -85,B 0,C 180,E1 7912.788,E2 7912.788} C_VEL
LIN {X 0,Y 317.412,Z 774.669,A -85,B 0,C 180,E1 7912.287,E2 7912.287} C_VEL
LIN {X 0,Y 310.66,Z 794.697,A -85,B 0,C 180,E1 7911.722,E2 7911.722} C_VEL
LIN {X 0,Y 301.724,Z 816.849,A -85,B 0,C 180,E1 7910.9,E2 7910.9} C_VEL
LIN {X 0,Y 291.935,Z 837.084,A -85,B 0,C 180,E1 7909.92,E2 7909.92} C_VEL
LIN {X 0,Y 279.963,Z 858.384,A -85,B 0,C 180,E1 7908.592,E2 7908.592} C_VEL
LIN {X 0,Y 268.17,Z 876.675,A -85,B 0,C 180,E1 7907.132,E2 7907.132} C_VEL
LIN {X 0,Y 254.299,Z 895.566,A -85,B 0,C 180,E1 7905.193,E2 7905.193} C_VEL
LIN {X 0,Y 240.496,Z 912.439,A -85,B 0,C 180,E1 7902.965,E2 7902.965} C_VEL
LIN {X 0,Y 226.202,Z 927.945,A -85,B 0,C 180,E1 7900.289,E2 7900.289} C_VEL
LIN {X 0,Y 211.704,Z 942.422,A -85,B 0,C 180,E1 7897.054,E2 7897.054} C_VEL
LIN {X 0,Y 197.234,Z 955.493,A -85,B 0,C 180,E1 7893.141,E2 7893.141} C_VEL
LIN {X 0,Y 182.461,Z 967.964,A -85,B 0,C 180,E1 7888.135,E2 7888.135} C_VEL
LIN {X 0,Y 169.835,Z 977.981,A -85,B 0,C 180,E1 7882.627,E2 7882.627} C_VEL
LIN {X 0,Y 157.435,Z 987.541,A -85,B 0,C 180,E1 7875.336,E2 7875.336} C_VEL
LIN {X 0,Y 148.422,Z 994.604,A -85,B 0,C 180,E1 7867.805,E2 7867.805} C_VEL
LIN {X 0,Y 141.399,Z 1000.525,A -85,B 0,C 180,E1 7858.738,E2 7858.738} C_VEL
LIN {X 0,Y 137.65,Z 1004.478,A -85,B 0,C 180,E1 7849.961,E2 7849.961} C_VEL
LIN {X 0,Y 136.152,Z 1006.949,A -85,B 0,C 180,E1 7841.007,E2 7841.007} C_VEL
LIN {X 0,Y 136.039,Z 1007.886,A -85,B 0,C 180,E1 7834.216,E2 7834.216} C_VEL
LIN {X 0,Y 136.072,Z 1008.032,A -85,B 0,C 180,E1 7828.317,E2 7828.317} C_VEL
LIN {X 0,Y 136.062,Z 1007.383,A -85,B 0,C 180,E1 7821.551,E2 7821.551} C_VEL
LIN {X 0,Y 136.767,Z 1005.663,A -85,B 0,C 180,E1 7813.874,E2 7813.874} C_VEL
LIN {X 0,Y 139.678,Z 1002.229,A -85,B 0,C 180,E1 7804.569,E2 7804.569} C_VEL
LIN {X 0,Y 145.308,Z 997.073,A -85,B 0,C 180,E1 7795.656,E2 7795.656} C_VEL
LIN {X 0,Y 154.168,Z 990.042,A -85,B 0,C 180,E1 7787.087,E2 7787.087} C_VEL
LIN {X 0,Y 164.847,Z 981.773,A -85,B 0,C 180,E1 7780.009,E2 7780.009} C_VEL
LIN {X 0,Y 178.5,Z 971.051,A -85,B 0,C 180,E1 7773.436,E2 7773.436} C_VEL
LIN {X 0,Y 192.145,Z 959.831,A -85,B 0,C 180,E1 7768.441,E2 7768.441} C_VEL
LIN {X 0,Y 207.024,Z 946.583,A -85,B 0,C 180,E1 7764.12,E2 7764.12} C_VEL
LIN {X 0,Y 222.166,Z 932.013,A -85,B 0,C 180,E1 7760.55,E2 7760.55} C_VEL
LIN {X 0,Y 236.576,Z 916.592,A -85,B 0,C 180,E1 7757.715,E2 7757.715} C_VEL
LIN {X 0,Y 251.727,Z 898.631,A -85,B 0,C 180,E1 7755.187,E2 7755.187} C_VEL
LIN {X 0,Y 264.655,Z 881.436,A -85,B 0,C 180,E1 7753.323,E2 7753.323} C_VEL
LIN {X 0,Y 277.665,Z 861.793,A -85,B 0,C 180,E1 7751.668,E2 7751.668} C_VEL
LIN {X 0,Y 289.312,Z 841.818,A -85,B 0,C 180,E1 7750.352,E2 7750.352} C_VEL
LIN {X 0,Y 299.507,Z 821.21,A -85,B 0,C 180,E1 7749.305,E2 7749.305} C_VEL
LIN {X 0,Y 308.295,Z 800.625,A -85,B 0,C 180,E1 7748.487,E2 7748.487} C_VEL
LIN {X 0,Y 315.622,Z 779.609,A -85,B 0,C 180,E1 7747.847,E2 7747.847} C_VEL
LIN {X 0,Y 322.103,Z 756.637,A -85,B 0,C 180,E1 7747.315,E2 7747.315} C_VEL
LIN {X 0,Y 326.741,Z 734.151,A -85,B 0,C 180,E1 7746.888,E2 7746.888} C_VEL
LIN {X 0,Y 330.882,Z 703.094,A -85,B 0,C 180,E1 7746.363,E2 7746.363} C_VEL
LIN {X 0,Y 340.518,Z 618.181,A -85,B 0,C 180,E1 7744.977,E2 7744.977} C_VEL
LIN {X 0,Y 339.606,Z 614.817,A -85,B 0,C 180,E1 7741.181,E2 7741.181} C_VEL
LIN {X 0,Y 339.649,Z 615.099,A -85,B 0,C 180,E1 7737.806,E2 7737.806} C_VEL
LIN {X 0,Y 340.454,Z 618.299,A -85,B 0,C 180,E1 7734.541,E2 7734.541} C_VEL
LIN {X 0,Y 328.142,Z 724.274,A -85,B 0,C 180,E1 7732.823,E2 7732.823} C_VEL
LIN {X 0,Y 323.718,Z 747.631,A -85,B 0,C 180,E1 7732.371,E2 7732.371} C_VEL
LIN {X 0,Y 318.151,Z 769.48,A -85,B 0,C 180,E1 7731.823,E2 7731.823} C_VEL
LIN {X 0,Y 310.916,Z 791.227,A -85,B 0,C 180,E1 7731.102,E2 7731.102} C_VEL
LIN {X 0,Y 302.335,Z 812.652,A -85,B 0,C 180,E1 7730.197,E2 7730.197} C_VEL
LIN {X 0,Y 292.68,Z 832.667,A -85,B 0,C 180,E1 7729.125,E2 7729.125} C_VEL
LIN {X 0,Y 280.826,Z 853.778,A -85,B 0,C 180,E1 7727.697,E2 7727.697} C_VEL
LIN {X 0,Y 269.242,Z 871.696,A -85,B 0,C 180,E1 7726.164,E2 7726.164} C_VEL
LIN {X 0,Y 255.638,Z 890.154,A -85,B 0,C 180,E1 7724.163,E2 7724.163} C_VEL
LIN {X 0,Y 241.947,Z 906.735,A -85,B 0,C 180,E1 7721.872,E2 7721.872} C_VEL
LIN {X 0,Y 227.847,Z 921.844,A -85,B 0,C 180,E1 7719.161,E2 7719.161} C_VEL
LIN {X 0,Y 213.534,Z 935.893,A -85,B 0,C 180,E1 7715.917,E2 7715.917} C_VEL
LIN {X 0,Y 199.218,Z 948.501,A -85,B 0,C 180,E1 7712.032,E2 7712.032} C_VEL
LIN {X 0,Y 184.566,Z 960.475,A -85,B 0,C 180,E1 7707.095,E2 7707.095} C_VEL
LIN {X 0,Y 171.978,Z 970.012,A -85,B 0,C 180,E1 7701.699,E2 7701.699} C_VEL
LIN {X 0,Y 159.493,Z 979.046,A -85,B 0,C 180,E1 7694.59,E2 7694.59} C_VEL
LIN {X 0,Y 149.892,Z 985.942,A -85,B 0,C 180,E1 7686.889,E2 7686.889} C_VEL
LIN {X 0,Y 142.59,Z 991.313,A -85,B 0,C 180,E1 7678.017,E2 7678.017} C_VEL
LIN {X 0,Y 138.334,Z 995.001,A -85,B 0,C 180,E1 7668.978,E2 7668.978} C_VEL
LIN {X 0,Y 136.506,Z 997.017,A -85,B 0,C 180,E1 7660.122,E2 7660.122} C_VEL
LIN {X 0,Y 136.098,Z 997.744,A -85,B 0,C 180,E1 7653.368,E2 7653.368} C_VEL
LIN {X 0,Y 136.092,Z 997.793,A -85,B 0,C 180,E1 7647.473,E2 7647.473} C_VEL
LIN {X 0,Y 136.394,Z 997.169,A -85,B 0,C 180,E1 7640.719,E2 7640.719} C_VEL
LIN {X 0,Y 137.807,Z 995.489,A -85,B 0,C 180,E1 7632.695,E2 7632.695} C_VEL
LIN {X 0,Y 141.81,Z 991.976,A -85,B 0,C 180,E1 7623.178,E2 7623.178} C_VEL
LIN {X 0,Y 147.996,Z 987.327,A -85,B 0,C 180,E1 7614.956,E2 7614.956} C_VEL
LIN {X 0,Y 157.496,Z 980.534,A -85,B 0,C 180,E1 7606.719,E2 7606.719} C_VEL
LIN {X 0,Y 168.422,Z 972.738,A -85,B 0,C 180,E1 7600.026,E2 7600.026} C_VEL
LIN {X 0,Y 181.186,Z 963.151,A -85,B 0,C 180,E1 7594.139,E2 7594.139} C_VEL
LIN {X 0,Y 195.308,Z 951.993,A -85,B 0,C 180,E1 7589.101,E2 7589.101} C_VEL
LIN {X 0,Y 209.586,Z 939.553,A -85,B 0,C 180,E1 7584.997,E2 7584.997} C_VEL
LIN {X 0,Y 224.523,Z 925.435,A -85,B 0,C 180,E1 7581.466,E2 7581.466} C_VEL
LIN {X 0,Y 238.494,Z 910.711,A -85,B 0,C 180,E1 7578.67,E2 7578.67} C_VEL
LIN {X 0,Y 253.824,Z 892.682,A -85,B 0,C 180,E1 7576.042,E2 7576.042} C_VEL
LIN {X 0,Y 266.954,Z 875.305,A -85,B 0,C 180,E1 7574.078,E2 7574.078} C_VEL
LIN {X 0,Y 279.468,Z 856.297,A -85,B 0,C 180,E1 7572.396,E2 7572.396} C_VEL
LIN {X 0,Y 290.791,Z 836.76,A -85,B 0,C 180,E1 7571.02,E2 7571.02} C_VEL
LIN {X 0,Y 300.714,Z 816.594,A -85,B 0,C 180,E1 7569.899,E2 7569.899} C_VEL
LIN {X 0,Y 309.697,Z 795.158,A -85,B 0,C 180,E1 7568.952,E2 7568.952} C_VEL
LIN {X 0,Y 316.463,Z 775.516,A -85,B 0,C 180,E1 7568.27,E2 7568.27} C_VEL
LIN {X 0,Y 322.827,Z 752.517,A -85,B 0,C 180,E1 7567.642,E2 7567.642} C_VEL
LIN {X 0,Y 327.254,Z 730.905,A -85,B 0,C 180,E1 7567.199,E2 7567.199} C_VEL
LIN {X 0,Y 331.386,Z 699.897,A -85,B 0,C 180,E1 7566.68,E2 7566.68} C_VEL
LIN {X 0,Y 340.671,Z 618.265,A -85,B 0,C 180,E1 7565.347,E2 7565.347} C_VEL
LIN {X 0,Y 339.798,Z 614.883,A -85,B 0,C 180,E1 7561.349,E2 7561.349} C_VEL
LIN {X 0,Y 339.841,Z 615.079,A -85,B 0,C 180,E1 7558.652,E2 7558.652} C_VEL
LIN {X 0,Y 340.708,Z 618.521,A -85,B 0,C 180,E1 7555.009,E2 7555.009} C_VEL
LIN {X 0,Y 336.443,Z 655.886,A -85,B 0,C 180,E1 7554.407,E2 7554.407} C_VEL
LIN {X 0,Y 335.461,Z 663.589,A -85,B 0,C 180,E1 7554.46,E2 7554.46} C_VEL
LIN {X 0,Y 332.512,Z 684.185,A -85,B 0,C 180,E1 7555.2,E2 7555.2} C_VEL
LIN {X 0,Y 331.687,Z 690.789,A -85,B 0,C 180,E1 7555.22,E2 7555.22} C_VEL
LIN {X 0,Y 326.741,Z 730.3,A -85,B 0,C 180,E1 7554.583,E2 7554.583} C_VEL
LIN {X 0,Y 322.104,Z 753.232,A -85,B 0,C 180,E1 7554.172,E2 7554.172} C_VEL
LIN {X 0,Y 315.307,Z 777.846,A -85,B 0,C 180,E1 7553.649,E2 7553.649} C_VEL
LIN {X 0,Y 308.568,Z 797.193,A -85,B 0,C 180,E1 7553.115,E2 7553.115} C_VEL
LIN {X 0,Y 299.124,Z 819.582,A -85,B 0,C 180,E1 7552.299,E2 7552.299} C_VEL
LIN {X 0,Y 288.973,Z 839.965,A -85,B 0,C 180,E1 7551.336,E2 7551.336} C_VEL
LIN {X 0,Y 277.067,Z 860.303,A -85,B 0,C 180,E1 7550.089,E2 7550.089} C_VEL
LIN {X 0,Y 264.174,Z 879.648,A -85,B 0,C 180,E1 7548.571,E2 7548.571} C_VEL
LIN {X 0,Y 250.599,Z 897.41,A -85,B 0,C 180,E1 7546.762,E2 7546.762} C_VEL
LIN {X 0,Y 235.575,Z 914.967,A -85,B 0,C 180,E1 7544.443,E2 7544.443} C_VEL
LIN {X 0,Y 221.054,Z 930.154,A -85,B 0,C 180,E1 7541.815,E2 7541.815} C_VEL
LIN {X 0,Y 205.36,Z 944.963,A -85,B 0,C 180,E1 7538.411,E2 7538.411} C_VEL
LIN {X 0,Y 190.561,Z 957.772,A -85,B 0,C 180,E1 7534.473,E2 7534.473} C_VEL
LIN {X 0,Y 176.011,Z 969.287,A -85,B 0,C 180,E1 7529.631,E2 7529.631} C_VEL
LIN {X 0,Y 162.41,Z 979.549,A -85,B 0,C 180,E1 7523.747,E2 7523.747} C_VEL
LIN {X 0,Y 150.119,Z 988.323,A -85,B 0,C 180,E1 7516.546,E2 7516.546} C_VEL
LIN {X 0,Y 139.959,Z 995.735,A -85,B 0,C 180,E1 7507.903,E2 7507.903} C_VEL
LIN {X 0,Y 133.413,Z 1000.865,A -85,B 0,C 180,E1 7499.15,E2 7499.15} C_VEL
LIN {X 0,Y 129.321,Z 1004.885,A -85,B 0,C 180,E1 7488.948,E2 7488.948} C_VEL
LIN {X 0,Y 128.121,Z 1006.868,A -85,B 0,C 180,E1 7480.34,E2 7480.34} C_VEL
LIN {X 0,Y 128.046,Z 1007.636,A -85,B 0,C 180,E1 7473.582,E2 7473.582} C_VEL
LIN {X 0,Y 128.065,Z 1007.708,A -85,B 0,C 180,E1 7467.764,E2 7467.764} C_VEL
LIN {X 0,Y 128.082,Z 1007.08,A -85,B 0,C 180,E1 7461.02,E2 7461.02} C_VEL
LIN {X 0,Y 128.927,Z 1005.356,A -85,B 0,C 180,E1 7452.864,E2 7452.864} C_VEL
LIN {X 0,Y 132.258,Z 1001.918,A -85,B 0,C 180,E1 7443.03,E2 7443.03} C_VEL
LIN {X 0,Y 138.505,Z 996.76,A -85,B 0,C 180,E1 7433.71,E2 7433.71} C_VEL
LIN {X 0,Y 148.14,Z 989.727,A -85,B 0,C 180,E1 7424.88,E2 7424.88} C_VEL
LIN {X 0,Y 159.405,Z 981.582,A -85,B 0,C 180,E1 7417.794,E2 7417.794} C_VEL
LIN {X 0,Y 174.014,Z 970.734,A -85,B 0,C 180,E1 7411.128,E2 7411.128} C_VEL
LIN {X 0,Y 188.629,Z 959.257,A -85,B 0,C 180,E1 7406.1,E2 7406.1} C_VEL
LIN {X 0,Y 203.749,Z 946.267,A -85,B 0,C 180,E1 7401.973,E2 7401.973} C_VEL
LIN {X 0,Y 218.586,Z 932.502,A -85,B 0,C 180,E1 7398.674,E2 7398.674} C_VEL
LIN {X 0,Y 233.821,Z 916.671,A -85,B 0,C 180,E1 7395.843,E2 7395.843} C_VEL
LIN {X 0,Y 248.913,Z 899.297,A -85,B 0,C 180,E1 7393.472,E2 7393.472} C_VEL
LIN {X 0,Y 261.923,Z 882.415,A -85,B 0,C 180,E1 7391.7,E2 7391.7} C_VEL
LIN {X 0,Y 275.709,Z 862.149,A -85,B 0,C 180,E1 7390.051,E2 7390.051} C_VEL
LIN {X 0,Y 287.322,Z 842.623,A -85,B 0,C 180,E1 7388.82,E2 7388.82} C_VEL
LIN {X 0,Y 297.691,Z 822.202,A -85,B 0,C 180,E1 7387.822,E2 7387.822} C_VEL
LIN {X 0,Y 306.932,Z 801.036,A -85,B 0,C 180,E1 7387.018,E2 7387.018} C_VEL
LIN {X 0,Y 314.431,Z 779.891,A -85,B 0,C 180,E1 7386.407,E2 7386.407} C_VEL
LIN {X 0,Y 320.979,Z 757.19,A -85,B 0,C 180,E1 7385.907,E2 7385.907} C_VEL
LIN {X 0,Y 325.754,Z 734.485,A -85,B 0,C 180,E1 7385.494,E2 7385.494} C_VEL
LIN {X 0,Y 329.984,Z 703.657,A -85,B 0,C 180,E1 7384.988,E2 7384.988} C_VEL
LIN {X 0,Y 339.053,Z 625.162,A -85,B 0,C 180,E1 7383.719,E2 7383.719} C_VEL
LIN {X 0,Y 338.609,Z 622.745,A -85,B 0,C 180,E1 7381.015,E2 7381.015} C_VEL
LIN {X 0,Y 338.649,Z 622.988,A -85,B 0,C 180,E1 7377.969,E2 7377.969} C_VEL
LIN {X 0,Y 339.006,Z 625.302,A -85,B 0,C 180,E1 7375.78,E2 7375.78} C_VEL
LIN {X 0,Y 327.238,Z 724.597,A -85,B 0,C 180,E1 7374.213,E2 7374.213} C_VEL
LIN {X 0,Y 322.752,Z 747.95,A -85,B 0,C 180,E1 7373.779,E2 7373.779} C_VEL
LIN {X 0,Y 317.11,Z 769.791,A -85,B 0,C 180,E1 7373.257,E2 7373.257} C_VEL
LIN {X 0,Y 309.932,Z 791.112,A -85,B 0,C 180,E1 7372.585,E2 7372.585} C_VEL
LIN {X 0,Y 301.539,Z 811.96,A -85,B 0,C 180,E1 7371.753,E2 7371.753} C_VEL
LIN {X 0,Y 291.683,Z 832.173,A -85,B 0,C 180,E1 7370.728,E2 7370.728} C_VEL
LIN {X 0,Y 280.641,Z 851.83,A -85,B 0,C 180,E1 7369.483,E2 7369.483} C_VEL
LIN {X 0,Y 268.774,Z 870.022,A -85,B 0,C 180,E1 7368.029,E2 7368.029} C_VEL
LIN {X 0,Y 255.17,Z 888.445,A -85,B 0,C 180,E1 7366.171,E2 7366.171} C_VEL
LIN {X 0,Y 242.127,Z 904.044,A -85,B 0,C 180,E1 7364.164,E2 7364.164} C_VEL
LIN {X 0,Y 226.738,Z 920.49,A -85,B 0,C 180,E1 7361.437,E2 7361.437} C_VEL
LIN {X 0,Y 212.489,Z 934.171,A -85,B 0,C 180,E1 7358.467,E2 7358.467} C_VEL
LIN {X 0,Y 197,Z 947.567,A -85,B 0,C 180,E1 7354.596,E2 7354.596} C_VEL
LIN {X 0,Y 182.315,Z 959.25,A -85,B 0,C 180,E1 7350.042,E2 7350.042} C_VEL
LIN {X 0,Y 168.227,Z 969.431,A -85,B 0,C 180,E1 7344.503,E2 7344.503} C_VEL
LIN {X 0,Y 155.31,Z 978.332,A -85,B 0,C 180,E1 7337.752,E2 7337.752} C_VEL
LIN {X 0,Y 145.064,Z 985.083,A -85,B 0,C 180,E1 7330.376,E2 7330.376} C_VEL
LIN {X 0,Y 136.272,Z 991.03,A -85,B 0,C 180,E1 7320.899,E2 7320.899} C_VEL
LIN {X 0,Y 131.304,Z 994.701,A -85,B 0,C 180,E1 7311.905,E2 7311.905} C_VEL
LIN {X 0,Y 128.735,Z 997.133,A -85,B 0,C 180,E1 7302.102,E2 7302.102} C_VEL
LIN {X 0,Y 128.132,Z 998.003,A -85,B 0,C 180,E1 7294.474,E2 7294.474} C_VEL
LIN {X 0,Y 128.099,Z 998.106,A -85,B 0,C 180,E1 7287.573,E2 7287.573} C_VEL
LIN {X 0,Y 128.408,Z 997.534,A -85,B 0,C 180,E1 7280.589,E2 7280.589} C_VEL
LIN {X 0,Y 129.812,Z 996.007,A -85,B 0,C 180,E1 7272.52,E2 7272.52} C_VEL
LIN {X 0,Y 134.03,Z 992.678,A -85,B 0,C 180,E1 7262.452,E2 7262.452} C_VEL
LIN {X 0,Y 140.567,Z 988.124,A -85,B 0,C 180,E1 7253.819,E2 7253.819} C_VEL
LIN {X 0,Y 151.076,Z 981.185,A -85,B 0,C 180,E1 7244.92,E2 7244.92} C_VEL
LIN {X 0,Y 162.62,Z 973.441,A -85,B 0,C 180,E1 7238.101,E2 7238.101} C_VEL
LIN {X 0,Y 176.674,Z 963.46,A -85,B 0,C 180,E1 7231.916,E2 7231.916} C_VEL
LIN {X 0,Y 190.909,Z 952.695,A -85,B 0,C 180,E1 7227.094,E2 7227.094} C_VEL
LIN {X 0,Y 205.447,Z 940.548,A -85,B 0,C 180,E1 7223.115,E2 7223.115} C_VEL
LIN {X 0,Y 220.82,Z 926.573,A -85,B 0,C 180,E1 7219.658,E2 7219.658} C_VEL
LIN {X 0,Y 235.141,Z 911.928,A -85,B 0,C 180,E1 7216.935,E2 7216.935} C_VEL
LIN {X 0,Y 249.927,Z 895.178,A -85,B 0,C 180,E1 7214.524,E2 7214.524} C_VEL
LIN {X 0,Y 263.046,Z 878.338,A -85,B 0,C 180,E1 7212.643,E2 7212.643} C_VEL
LIN {X 0,Y 276.449,Z 858.81,A -85,B 0,C 180,E1 7210.931,E2 7210.931} C_VEL
LIN {X 0,Y 287.5,Z 840.364,A -85,B 0,C 180,E1 7209.653,E2 7209.653} C_VEL
LIN {X 0,Y 298.208,Z 819.505,A -85,B 0,C 180,E1 7208.507,E2 7208.507} C_VEL
LIN {X 0,Y 307.284,Z 798.789,A -85,B 0,C 180,E1 7207.605,E2 7207.605} C_VEL
LIN {X 0,Y 314.906,Z 777.368,A -85,B 0,C 180,E1 7206.874,E2 7206.874} C_VEL
LIN {X 0,Y 321.296,Z 755.265,A -85,B 0,C 180,E1 7206.282,E2 7206.282} C_VEL
LIN {X 0,Y 326.075,Z 732.673,A -85,B 0,C 180,E1 7205.831,E2 7205.831} C_VEL
LIN {X 0,Y 330.019,Z 704.784,A -85,B 0,C 180,E1 7205.374,E2 7205.374} C_VEL
LIN {X 0,Y 339.233,Z 625.225,A -85,B 0,C 180,E1 7204.099,E2 7204.099} C_VEL
LIN {X 0,Y 338.823,Z 622.824,A -85,B 0,C 180,E1 7201.353,E2 7201.353} C_VEL
LIN {X 0,Y 338.847,Z 622.968,A -85,B 0,C 180,E1 7198.817,E2 7198.817} C_VEL
LIN {X 0,Y 339.238,Z 625.646,A -85,B 0,C 180,E1 7196.245,E2 7196.245} C_VEL
LIN {X 0,Y 331.687,Z 690.789,A -85,B 0,C 180,E1 7195.22,E2 7195.22} C_VEL
LIN {X 0,Y 330.724,Z 698.487,A -85,B 0,C 180,E1 7195.27,E2 7195.27} C_VEL
LIN {X 0,Y 327.725,Z 719.06,A -85,B 0,C 180,E1 7196.04,E2 7196.04} C_VEL
LIN {X 0,Y 326.742,Z 725.65,A -85,B 0,C 180,E1 7196.061,E2 7196.061} C_VEL
LIN {X 0,Y 322.127,Z 749.754,A -85,B 0,C 180,E1 7195.656,E2 7195.656} C_VEL
